LIN {X 0,Y 517.937,Z 91.598,A -85,B 0,C 180,E1 -4909.404,E2 -4909.404} C_VEL
LIN {X 0,Y 516.923,Z 91.726,A -85,B 0,C 180,E1 -4910.052,E2 -4910.052} C_VEL
LIN {X 0,Y 516.851,Z 91.735,A -85,B 0,C 180,E1 -4910.271,E2 -4910.271} C_VEL
LIN {X 0,Y 516.906,Z 91.845,A -85,B 0,C 180,E1 -4911.136,E2 -4911.136} C_VEL
LIN {X 0,Y 518.401,Z 99.769,A -85,B 0,C 180,E1 -4912.604,E2 -4912.604} C_VEL
LIN {X 0,Y 518.069,Z 113.892,A -85,B 0,C 180,E1 -4915.029,E2 -4915.029} C_VEL
LIN {X 0,Y 518.021,Z 116.431,A -85,B 0,C 180,E1 -4915.437,E2 -4915.437} C_VEL
LIN {X 0,Y 520.471,Z 128.644,A -85,B 0,C 180,E1 -4915.705,E2 -4915.705} C_VEL
LIN {X 0,Y 519.69,Z 253.321,A -85,B 0,C 180,E1 -4917.481,E2 -4917.481} C_VEL
LIN {X 0,Y 519.462,Z 267.315,A -85,B 0,C 180,E1 -4917.838,E2 -4917.838} C_VEL
LIN {X 0,Y 519.171,Z 280.563,A -85,B 0,C 180,E1 -4918.326,E2 -4918.326} C_VEL
LIN {X 0,Y 518.764,Z 294.503,A -85,B 0,C 180,E1 -4919.014,E2 -4919.014} C_VEL
LIN {X 0,Y 518.356,Z 306.612,A -85,B 0,C 180,E1 -4919.777,E2 -4919.777} C_VEL
LIN {X 0,Y 517.938,Z 319.149,A -85,B 0,C 180,E1 -4920.758,E2 -4920.758} C_VEL
LIN {X 0,Y 517.552,Z 330.416,A -85,B 0,C 180,E1 -4921.842,E2 -4921.842} C_VEL
LIN {X 0,Y 517.178,Z 339.685,A -85,B 0,C 180,E1 -4922.919,E2 -4922.919} C_VEL
LIN {X 0,Y 516.871,Z 348.845,A -85,B 0,C 180,E1 -4924.207,E2 -4924.207} C_VEL
LIN {X 0,Y 516.661,Z 355.972,A -85,B 0,C 180,E1 -4925.418,E2 -4925.418} C_VEL
LIN {X 0,Y 516.507,Z 362.417,A -85,B 0,C 180,E1 -4926.758,E2 -4926.758} C_VEL
LIN {X 0,Y 516.393,Z 367.484,A -85,B 0,C 180,E1 -4928.075,E2 -4928.075} C_VEL
LIN {X 0,Y 516.349,Z 371.085,A -85,B 0,C 180,E1 -4929.274,E2 -4929.274} C_VEL
LIN {X 0,Y 516.314,Z 373.093,A -85,B 0,C 180,E1 -4930.104,E2 -4930.104} C_VEL
LIN {X 0,Y 516.164,Z 375.912,A -85,B 0,C 180,E1 -4931.749,E2 -4931.749} C_VEL
LIN {X 0,Y 516.203,Z 376.744,A -85,B 0,C 180,E1 -4932.57,E2 -4932.57} C_VEL
LIN {X 0,Y 516.155,Z 377.306,A -85,B 0,C 180,E1 -4934.197,E2 -4934.197} C_VEL
LIN {X 0,Y 516.205,Z 376.454,A -85,B 0,C 180,E1 -4935.813,E2 -4935.813} C_VEL
LIN {X 0,Y 516.269,Z 374.205,A -85,B 0,C 180,E1 -4937.419,E2 -4937.419} C_VEL
LIN {X 0,Y 516.334,Z 370.533,A -85,B 0,C 180,E1 -4939.014,E2 -4939.014} C_VEL
LIN {X 0,Y 516.397,Z 365.356,A -85,B 0,C 180,E1 -4940.6,E2 -4940.6} C_VEL
LIN {X 0,Y 516.526,Z 360.334,A -85,B 0,C 180,E1 -4941.785,E2 -4941.785} C_VEL
LIN {X 0,Y 516.761,Z 353.621,A -85,B 0,C 180,E1 -4943.085,E2 -4943.085} C_VEL
LIN {X 0,Y 516.944,Z 345.726,A -85,B 0,C 180,E1 -4944.342,E2 -4944.342} C_VEL
LIN {X 0,Y 517.288,Z 336.792,A -85,B 0,C 180,E1 -4945.518,E2 -4945.518} C_VEL
LIN {X 0,Y 517.677,Z 326.031,A -85,B 0,C 180,E1 -4946.691,E2 -4946.691} C_VEL
LIN {X 0,Y 518.065,Z 315.147,A -85,B 0,C 180,E1 -4947.666,E2 -4947.666} C_VEL
LIN {X 0,Y 518.475,Z 303.235,A -85,B 0,C 180,E1 -4948.543,E2 -4948.543} C_VEL
LIN {X 0,Y 518.925,Z 289.938,A -85,B 0,C 180,E1 -4949.32,E2 -4949.32} C_VEL
LIN {X 0,Y 519.246,Z 277.171,A -85,B 0,C 180,E1 -4949.902,E2 -4949.902} C_VEL
LIN {X 0,Y 519.516,Z 263.525,A -85,B 0,C 180,E1 -4950.362,E2 -4950.362} C_VEL
LIN {X 0,Y 519.652,Z 249.563,A -85,B 0,C 180,E1 -4950.677,E2 -4950.677} C_VEL
LIN {X 0,Y 520.387,Z 127.623,A -85,B 0,C 180,E1 -4952.399,E2 -4952.399} C_VEL
LIN {X 0,Y 517.972,Z 116.11,A -85,B 0,C 180,E1 -4952.66,E2 -4952.66} C_VEL
LIN {X 0,Y 518.473,Z 99.766,A -85,B 0,C 180,E1 -4955.444,E2 -4955.444} C_VEL
LIN {X 0,Y 516.971,Z 91.715,A -85,B 0,C 180,E1 -4956.925,E2 -4956.925} C_VEL
LIN {X 0,Y 516.932,Z 91.719,A -85,B 0,C 180,E1 -4959.388,E2 -4959.388} C_VEL
LIN {X 0,Y 516.933,Z 91.719,A -85,B 0,C 180,E1 -4962.563,E2 -4962.563} C_VEL
LIN {X 0,Y 516.94,Z 91.715,A -85,B 0,C 180,E1 -4965.161,E2 -4965.161} C_VEL
LIN {X 0,Y 516.893,Z 91.72,A -85,B 0,C 180,E1 -4968.222,E2 -4968.222} C_VEL
LIN {X 0,Y 516.882,Z 91.72,A -85,B 0,C 180,E1 -4970.701,E2 -4970.701} C_VEL
LIN {X 0,Y 516.878,Z 91.726,A -85,B 0,C 180,E1 -4973.222,E2 -4973.222} C_VEL
LIN {X 0,Y 516.917,Z 91.716,A -85,B 0,C 180,E1 -4976.2,E2 -4976.2} C_VEL
LIN {X 0,Y 516.906,Z 91.725,A -85,B 0,C 180,E1 -4979.304,E2 -4979.304} C_VEL
LIN {X 0,Y 516.875,Z 91.722,A -85,B 0,C 180,E1 -4982.548,E2 -4982.548} C_VEL
LIN {X 0,Y 516.884,Z 91.724,A -85,B 0,C 180,E1 -4985.34,E2 -4985.34} C_VEL
LIN {X 0,Y 516.886,Z 91.725,A -85,B 0,C 180,E1 -4988.714,E2 -4988.714} C_VEL
LIN {X 0,Y 516.893,Z 91.719,A -85,B 0,C 180,E1 -4991.775,E2 -4991.775} C_VEL
LIN {X 0,Y 516.889,Z 91.724,A -85,B 0,C 180,E1 -4995.012,E2 -4995.012} C_VEL
LIN {X 0,Y 516.886,Z 91.721,A -85,B 0,C 180,E1 -4997.24,E2 -4997.24} C_VEL
LIN {X 0,Y 516.905,Z 91.722,A -85,B 0,C 180,E1 -5000.286,E2 -5000.286} C_VEL
LIN {X 0,Y 516.862,Z 91.723,A -85,B 0,C 180,E1 -5003.343,E2 -5003.343} C_VEL
LIN {X 0,Y 516.888,Z 91.724,A -85,B 0,C 180,E1 -5006.124,E2 -5006.124} C_VEL
LIN {X 0,Y 516.871,Z 91.723,A -85,B 0,C 180,E1 -5008.937,E2 -5008.937} C_VEL
LIN {X 0,Y 516.901,Z 91.719,A -85,B 0,C 180,E1 -5011.588,E2 -5011.588} C_VEL
LIN {X 0,Y 516.915,Z 91.724,A -85,B 0,C 180,E1 -5014.214,E2 -5014.214} C_VEL
LIN {X 0,Y 516.888,Z 91.72,A -85,B 0,C 180,E1 -5016.781,E2 -5016.781} C_VEL
LIN {X 0,Y 516.919,Z 91.721,A -85,B 0,C 180,E1 -5019.734,E2 -5019.734} C_VEL
LIN {X 0,Y 516.913,Z 91.717,A -85,B 0,C 180,E1 -5022.599,E2 -5022.599} C_VEL
LIN {X 0,Y 516.924,Z 91.715,A -85,B 0,C 180,E1 -5025.033,E2 -5025.033} C_VEL
LIN {X 0,Y 516.988,Z 91.709,A -85,B 0,C 180,E1 -5028.237,E2 -5028.237} C_VEL
LIN {X 0,Y 516.96,Z 91.716,A -85,B 0,C 180,E1 -5031.402,E2 -5031.402} C_VEL
LIN {X 0,Y 517.034,Z 91.701,A -85,B 0,C 180,E1 -5034.543,E2 -5034.543} C_VEL
LIN {X 0,Y 517.074,Z 91.701,A -85,B 0,C 180,E1 -5037.666,E2 -5037.666} C_VEL
LIN {X 0,Y 517.087,Z 91.696,A -85,B 0,C 180,E1 -5040.781,E2 -5040.781} C_VEL
LIN {X 0,Y 517.008,Z 91.711,A -85,B 0,C 180,E1 -5043.119,E2 -5043.119} C_VEL
LIN {X 0,Y 517.002,Z 91.705,A -85,B 0,C 180,E1 -5046.246,E2 -5046.246} C_VEL
LIN {X 0,Y 516.947,Z 91.716,A -85,B 0,C 180,E1 -5049.392,E2 -5049.392} C_VEL
LIN {X 0,Y 516.945,Z 91.712,A -85,B 0,C 180,E1 -5051.81,E2 -5051.81} C_VEL
LIN {X 0,Y 516.938,Z 91.718,A -85,B 0,C 180,E1 -5055.149,E2 -5055.149} C_VEL
LIN {X 0,Y 516.92,Z 91.717,A -85,B 0,C 180,E1 -5058.224,E2 -5058.224} C_VEL
LIN {X 0,Y 516.907,Z 91.726,A -85,B 0,C 180,E1 -5060.704,E2 -5060.704} C_VEL
LIN {X 0,Y 516.907,Z 91.719,A -85,B 0,C 180,E1 -5064.074,E2 -5064.074} C_VEL
LIN {X 0,Y 516.926,Z 91.721,A -85,B 0,C 180,E1 -5066.66,E2 -5066.66} C_VEL
LIN {X 0,Y 516.908,Z 91.717,A -85,B 0,C 180,E1 -5069.526,E2 -5069.526} C_VEL
LIN {X 0,Y 516.895,Z 91.724,A -85,B 0,C 180,E1 -5072.546,E2 -5072.546} C_VEL
LIN {X 0,Y 516.876,Z 91.721,A -85,B 0,C 180,E1 -5075.334,E2 -5075.334} C_VEL
LIN {X 0,Y 516.878,Z 91.726,A -85,B 0,C 180,E1 -5077.945,E2 -5077.945} C_VEL
LIN {X 0,Y 516.882,Z 91.721,A -85,B 0,C 180,E1 -5080.743,E2 -5080.743} C_VEL
LIN {X 0,Y 516.883,Z 91.72,A -85,B 0,C 180,E1 -5082.833,E2 -5082.833} C_VEL
LIN {X 0,Y 516.922,Z 91.715,A -85,B 0,C 180,E1 -5085.012,E2 -5085.012} C_VEL
LIN {X 0,Y 516.914,Z 91.718,A -85,B 0,C 180,E1 -5088.4,E2 -5088.4} C_VEL
LIN {X 0,Y 516.88,Z 91.723,A -85,B 0,C 180,E1 -5091.286,E2 -5091.286} C_VEL
LIN {X 0,Y 516.871,Z 91.723,A -85,B 0,C 180,E1 -5094.221,E2 -5094.221} C_VEL
LIN {X 0,Y 516.895,Z 91.721,A -85,B 0,C 180,E1 -5097.055,E2 -5097.055} C_VEL
LIN {X 0,Y 516.887,Z 91.726,A -85,B 0,C 180,E1 -5099.797,E2 -5099.797} C_VEL
LIN {X 0,Y 516.926,Z 91.719,A -85,B 0,C 180,E1 -5102.469,E2 -5102.469} C_VEL
LIN {X 0,Y 516.957,Z 91.852,A -85,B 0,C 180,E1 -5103.888,E2 -5103.888} C_VEL
LIN {X 0,Y 519.076,Z 102.657,A -85,B 0,C 180,E1 -5105.611,E2 -5105.611} C_VEL
LIN {X 0,Y 518.535,Z 121.144,A -85,B 0,C 180,E1 -5108.327,E2 -5108.327} C_VEL
LIN {X 0,Y 517.999,Z 142.503,A -85,B 0,C 180,E1 -5111.381,E2 -5111.381} C_VEL
LIN {X 0,Y 520.393,Z 156.779,A -85,B 0,C 180,E1 -5111.672,E2 -5111.672} C_VEL
LIN {X 0,Y 519.58,Z 280.355,A -85,B 0,C 180,E1 -5113.423,E2 -5113.423} C_VEL
LIN {X 0,Y 519.338,Z 294.907,A -85,B 0,C 180,E1 -5113.792,E2 -5113.792} C_VEL
LIN {X 0,Y 519.05,Z 308.369,A -85,B 0,C 180,E1 -5114.289,E2 -5114.289} C_VEL
LIN {X 0,Y 518.646,Z 320.6,A -85,B 0,C 180,E1 -5114.881,E2 -5114.881} C_VEL
LIN {X 0,Y 518.226,Z 333.464,A -85,B 0,C 180,E1 -5115.672,E2 -5115.672} C_VEL
LIN {X 0,Y 517.779,Z 345.158,A -85,B 0,C 180,E1 -5116.56,E2 -5116.56} C_VEL
LIN {X 0,Y 517.474,Z 354.895,A -85,B 0,C 180,E1 -5117.451,E2 -5117.451} C_VEL
LIN {X 0,Y 517.116,Z 365.679,A -85,B 0,C 180,E1 -5118.636,E2 -5118.636} C_VEL
LIN {X 0,Y 516.817,Z 374.585,A -85,B 0,C 180,E1 -5119.819,E2 -5119.819} C_VEL
LIN {X 0,Y 516.607,Z 383.12,A -85,B 0,C 180,E1 -5121.198,E2 -5121.198} C_VEL
LIN {X 0,Y 516.443,Z 389.998,A -85,B 0,C 180,E1 -5122.573,E2 -5122.573} C_VEL
LIN {X 0,Y 516.352,Z 396.142,A -85,B 0,C 180,E1 -5124.142,E2 -5124.142} C_VEL
LIN {X 0,Y 516.262,Z 399.65,A -85,B 0,C 180,E1 -5125.316,E2 -5125.316} C_VEL
LIN {X 0,Y 516.325,Z 401.539,A -85,B 0,C 180,E1 -5126.099,E2 -5126.099} C_VEL
LIN {X 0,Y 516.26,Z 404.245,A -85,B 0,C 180,E1 -5127.661,E2 -5127.661} C_VEL
LIN {X 0,Y 516.158,Z 405.582,A -85,B 0,C 180,E1 -5129.221,E2 -5129.221} C_VEL
LIN {X 0,Y 516.158,Z 405.579,A -85,B 0,C 180,E1 -5130.781,E2 -5130.781} C_VEL
LIN {X 0,Y 516.261,Z 404.237,A -85,B 0,C 180,E1 -5132.342,E2 -5132.342} C_VEL
LIN {X 0,Y 516.325,Z 401.526,A -85,B 0,C 180,E1 -5133.904,E2 -5133.904} C_VEL
LIN {X 0,Y 516.354,Z 397.368,A -85,B 0,C 180,E1 -5135.468,E2 -5135.468} C_VEL
LIN {X 0,Y 516.405,Z 391.641,A -85,B 0,C 180,E1 -5137.037,E2 -5137.037} C_VEL
LIN {X 0,Y 516.562,Z 385.188,A -85,B 0,C 180,E1 -5138.411,E2 -5138.411} C_VEL
LIN {X 0,Y 516.752,Z 377.171,A -85,B 0,C 180,E1 -5139.789,E2 -5139.789} C_VEL
LIN {X 0,Y 517.05,Z 368.787,A -85,B 0,C 180,E1 -5140.971,E2 -5140.971} C_VEL
LIN {X 0,Y 517.371,Z 358.473,A -85,B 0,C 180,E1 -5142.18,E2 -5142.18} C_VEL
LIN {X 0,Y 517.722,Z 347.43,A -85,B 0,C 180,E1 -5143.244,E2 -5143.244} C_VEL
LIN {X 0,Y 518.078,Z 336.228,A -85,B 0,C 180,E1 -5144.134,E2 -5144.134} C_VEL
LIN {X 0,Y 518.512,Z 324.028,A -85,B 0,C 180,E1 -5144.925,E2 -5144.925} C_VEL
LIN {X 0,Y 518.956,Z 310.488,A -85,B 0,C 180,E1 -5145.615,E2 -5145.615} C_VEL
LIN {X 0,Y 519.26,Z 296.705,A -85,B 0,C 180,E1 -5146.147,E2 -5146.147} C_VEL
LIN {X 0,Y 519.549,Z 282.425,A -85,B 0,C 180,E1 -5146.53,E2 -5146.53} C_VEL
LIN {X 0,Y 519.768,Z 258.348,A -85,B 0,C 180,E1 -5146.902,E2 -5146.902} C_VEL
LIN {X 0,Y 520.277,Z 155.65,A -85,B 0,C 180,E1 -5148.347,E2 -5148.347} C_VEL
LIN {X 0,Y 517.932,Z 142.086,A -85,B 0,C 180,E1 -5148.637,E2 -5148.637} C_VEL
LIN {X 0,Y 518.551,Z 121.098,A -85,B 0,C 180,E1 -5151.675,E2 -5151.675} C_VEL
LIN {X 0,Y 519.092,Z 102.719,A -85,B 0,C 180,E1 -5154.391,E2 -5154.391} C_VEL
LIN {X 0,Y 517.157,Z 92.942,A -85,B 0,C 180,E1 -5155.975,E2 -5155.975} C_VEL
LIN {X 0,Y 516.91,Z 91.724,A -85,B 0,C 180,E1 -5156.187,E2 -5156.187} C_VEL
LIN {X 0,Y 516.925,Z 91.723,A -85,B 0,C 180,E1 -5158.416,E2 -5158.416} C_VEL
LIN {X 0,Y 516.898,Z 91.724,A -85,B 0,C 180,E1 -5161.11,E2 -5161.11} C_VEL
LIN {X 0,Y 516.897,Z 91.727,A -85,B 0,C 180,E1 -5163.963,E2 -5163.963} C_VEL
LIN {X 0,Y 516.864,Z 91.724,A -85,B 0,C 180,E1 -5166.748,E2 -5166.748} C_VEL
LIN {X 0,Y 516.883,Z 91.726,A -85,B 0,C 180,E1 -5169.722,E2 -5169.722} C_VEL
LIN {X 0,Y 516.918,Z 91.72,A -85,B 0,C 180,E1 -5171.776,E2 -5171.776} C_VEL
LIN {X 0,Y 516.908,Z 91.718,A -85,B 0,C 180,E1 -5175.007,E2 -5175.007} C_VEL
LIN {X 0,Y 516.926,Z 91.71,A -85,B 0,C 180,E1 -5178.399,E2 -5178.399} C_VEL
LIN {X 0,Y 516.889,Z 91.724,A -85,B 0,C 180,E1 -5181.283,E2 -5181.283} C_VEL
LIN {X 0,Y 516.88,Z 91.722,A -85,B 0,C 180,E1 -5184.219,E2 -5184.219} C_VEL
LIN {X 0,Y 516.894,Z 91.722,A -85,B 0,C 180,E1 -5187.051,E2 -5187.051} C_VEL
LIN {X 0,Y 516.896,Z 91.722,A -85,B 0,C 180,E1 -5189.795,E2 -5189.795} C_VEL
LIN {X 0,Y 516.906,Z 91.716,A -85,B 0,C 180,E1 -5192.464,E2 -5192.464} C_VEL
LIN {X 0,Y 516.878,Z 91.728,A -85,B 0,C 180,E1 -5195.068,E2 -5195.068} C_VEL
LIN {X 0,Y 516.882,Z 91.722,A -85,B 0,C 180,E1 -5197.62,E2 -5197.62} C_VEL
LIN {X 0,Y 516.942,Z 91.71,A -85,B 0,C 180,E1 -5200.128,E2 -5200.128} C_VEL
LIN {X 0,Y 516.907,Z 91.723,A -85,B 0,C 180,E1 -5202.593,E2 -5202.593} C_VEL
LIN {X 0,Y 516.947,Z 91.717,A -85,B 0,C 180,E1 -5205.028,E2 -5205.028} C_VEL
LIN {X 0,Y 516.978,Z 91.711,A -85,B 0,C 180,E1 -5208.232,E2 -5208.232} C_VEL
LIN {X 0,Y 516.963,Z 91.71,A -85,B 0,C 180,E1 -5211.397,E2 -5211.397} C_VEL
LIN {X 0,Y 517.021,Z 91.709,A -85,B 0,C 180,E1 -5214.538,E2 -5214.538} C_VEL
LIN {X 0,Y 517.088,Z 91.694,A -85,B 0,C 180,E1 -5217.661,E2 -5217.661} C_VEL
LIN {X 0,Y 517.096,Z 91.692,A -85,B 0,C 180,E1 -5220.776,E2 -5220.776} C_VEL
LIN {X 0,Y 516.988,Z 91.708,A -85,B 0,C 180,E1 -5223.114,E2 -5223.114} C_VEL
LIN {X 0,Y 516.993,Z 91.711,A -85,B 0,C 180,E1 -5226.241,E2 -5226.241} C_VEL
LIN {X 0,Y 516.944,Z 91.715,A -85,B 0,C 180,E1 -5229.386,E2 -5229.386} C_VEL
LIN {X 0,Y 516.954,Z 91.718,A -85,B 0,C 180,E1 -5231.804,E2 -5231.804} C_VEL
LIN {X 0,Y 516.943,Z 91.716,A -85,B 0,C 180,E1 -5235.142,E2 -5235.142} C_VEL
LIN {X 0,Y 516.91,Z 91.718,A -85,B 0,C 180,E1 -5238.219,E2 -5238.219} C_VEL
LIN {X 0,Y 516.901,Z 91.718,A -85,B 0,C 180,E1 -5240.698,E2 -5240.698} C_VEL
LIN {X 0,Y 516.88,Z 91.721,A -85,B 0,C 180,E1 -5244.07,E2 -5244.07} C_VEL
LIN {X 0,Y 516.9,Z 91.72,A -85,B 0,C 180,E1 -5246.655,E2 -5246.655} C_VEL
LIN {X 0,Y 516.899,Z 91.715,A -85,B 0,C 180,E1 -5249.52,E2 -5249.52} C_VEL
LIN {X 0,Y 516.882,Z 91.725,A -85,B 0,C 180,E1 -5252.539,E2 -5252.539} C_VEL
LIN {X 0,Y 516.852,Z 91.728,A -85,B 0,C 180,E1 -5255.326,E2 -5255.326} C_VEL
LIN {X 0,Y 516.863,Z 91.721,A -85,B 0,C 180,E1 -5257.939,E2 -5257.939} C_VEL
LIN {X 0,Y 516.867,Z 91.727,A -85,B 0,C 180,E1 -5260.738,E2 -5260.738} C_VEL
LIN {X 0,Y 516.864,Z 91.729,A -85,B 0,C 180,E1 -5262.828,E2 -5262.828} C_VEL
LIN {X 0,Y 516.875,Z 91.724,A -85,B 0,C 180,E1 -5265.004,E2 -5265.004} C_VEL
LIN {X 0,Y 516.88,Z 91.731,A -85,B 0,C 180,E1 -5268.397,E2 -5268.397} C_VEL
LIN {X 0,Y 516.851,Z 91.735,A -85,B 0,C 180,E1 -5270.271,E2 -5270.271} C_VEL
LIN {X 0,Y 516.63,Z 92.161,A -85,B 0,C 180,E1 -5270.7,E2 -5270.7} C_VEL
LIN {X 0,Y 516.043,Z 93.272,A -85,B 0,C 180,E1 -5271.112,E2 -5271.112} C_VEL
LIN {X 0,Y 514.758,Z 95.823,A -85,B 0,C 180,E1 -5271.695,E2 -5271.695} C_VEL
LIN {X 0,Y 511.765,Z 103.822,A -85,B 0,C 180,E1 -5272.982,E2 -5272.982} C_VEL
LIN {X 0,Y 511.44,Z 106.048,A -85,B 0,C 180,E1 -5273.361,E2 -5273.361} C_VEL
LIN {X 0,Y 511.096,Z 116.359,A -85,B 0,C 180,E1 -5275.149,E2 -5275.149} C_VEL
LIN {X 0,Y 513.748,Z 129.088,A -85,B 0,C 180,E1 -5275.457,E2 -5275.457} C_VEL
LIN {X 0,Y 512.927,Z 252.499,A -85,B 0,C 180,E1 -5277.232,E2 -5277.232} C_VEL
LIN {X 0,Y 512.654,Z 267.254,A -85,B 0,C 180,E1 -5277.606,E2 -5277.606} C_VEL
LIN {X 0,Y 512.346,Z 280.832,A -85,B 0,C 180,E1 -5278.113,E2 -5278.113} C_VEL
LIN {X 0,Y 511.918,Z 294.283,A -85,B 0,C 180,E1 -5278.783,E2 -5278.783} C_VEL
LIN {X 0,Y 511.462,Z 307.149,A -85,B 0,C 180,E1 -5279.605,E2 -5279.605} C_VEL
LIN {X 0,Y 511.042,Z 319.053,A -85,B 0,C 180,E1 -5280.55,E2 -5280.55} C_VEL
LIN {X 0,Y 510.64,Z 329.18,A -85,B 0,C 180,E1 -5281.525,E2 -5281.525} C_VEL
LIN {X 0,Y 510.19,Z 339.675,A -85,B 0,C 180,E1 -5282.739,E2 -5282.739} C_VEL
LIN {X 0,Y 509.867,Z 348.887,A -85,B 0,C 180,E1 -5284.045,E2 -5284.045} C_VEL
LIN {X 0,Y 509.615,Z 356.504,A -85,B 0,C 180,E1 -5285.365,E2 -5285.365} C_VEL
LIN {X 0,Y 509.432,Z 363.378,A -85,B 0,C 180,E1 -5286.846,E2 -5286.846} C_VEL
LIN {X 0,Y 509.319,Z 368.114,A -85,B 0,C 180,E1 -5288.125,E2 -5288.125} C_VEL
LIN {X 0,Y 509.233,Z 372.697,A -85,B 0,C 180,E1 -5289.785,E2 -5289.785} C_VEL
LIN {X 0,Y 509.087,Z 375.784,A -85,B 0,C 180,E1 -5291.486,E2 -5291.486} C_VEL
LIN {X 0,Y 509.08,Z 377.3,A -85,B 0,C 180,E1 -5293.146,E2 -5293.146} C_VEL
LIN {X 0,Y 509.091,Z 377.376,A -85,B 0,C 180,E1 -5294.793,E2 -5294.793} C_VEL
LIN {X 0,Y 509.108,Z 376.02,A -85,B 0,C 180,E1 -5296.426,E2 -5296.426} C_VEL
LIN {X 0,Y 509.205,Z 373.247,A -85,B 0,C 180,E1 -5298.051,E2 -5298.051} C_VEL
LIN {X 0,Y 509.291,Z 369.024,A -85,B 0,C 180,E1 -5299.664,E2 -5299.664} C_VEL
LIN {X 0,Y 509.418,Z 363.242,A -85,B 0,C 180,E1 -5301.27,E2 -5301.27} C_VEL
LIN {X 0,Y 509.621,Z 356.741,A -85,B 0,C 180,E1 -5302.67,E2 -5302.67} C_VEL
LIN {X 0,Y 509.885,Z 348.713,A -85,B 0,C 180,E1 -5304.065,E2 -5304.065} C_VEL
LIN {X 0,Y 510.187,Z 340.337,A -85,B 0,C 180,E1 -5305.258,E2 -5305.258} C_VEL
LIN {X 0,Y 510.597,Z 330.264,A -85,B 0,C 180,E1 -5306.448,E2 -5306.448} C_VEL
LIN {X 0,Y 510.983,Z 319.057,A -85,B 0,C 180,E1 -5307.536,E2 -5307.536} C_VEL
LIN {X 0,Y 511.402,Z 307.943,A -85,B 0,C 180,E1 -5308.424,E2 -5308.424} C_VEL
LIN {X 0,Y 511.893,Z 295.811,A -85,B 0,C 180,E1 -5309.212,E2 -5309.212} C_VEL
LIN {X 0,Y 512.29,Z 282.406,A -85,B 0,C 180,E1 -5309.901,E2 -5309.901} C_VEL
LIN {X 0,Y 512.615,Z 268.364,A -85,B 0,C 180,E1 -5310.441,E2 -5310.441} C_VEL
LIN {X 0,Y 512.823,Z 254.558,A -85,B 0,C 180,E1 -5310.809,E2 -5310.809} C_VEL
LIN {X 0,Y 513.055,Z 227.07,A -85,B 0,C 180,E1 -5311.231,E2 -5311.231} C_VEL
LIN {X 0,Y 513.653,Z 128.738,A -85,B 0,C 180,E1 -5312.633,E2 -5312.633} C_VEL
LIN {X 0,Y 511.048,Z 116.22,A -85,B 0,C 180,E1 -5312.931,E2 -5312.931} C_VEL
LIN {X 0,Y 511.553,Z 101.194,A -85,B 0,C 180,E1 -5315.517,E2 -5315.517} C_VEL
LIN {X 0,Y 509.951,Z 92.59,A -85,B 0,C 180,E1 -5317.124,E2 -5317.124} C_VEL
LIN {X 0,Y 509.874,Z 92.6,A -85,B 0,C 180,E1 -5319.52,E2 -5319.52} C_VEL
LIN {X 0,Y 509.912,Z 92.598,A -85,B 0,C 180,E1 -5321.93,E2 -5321.93} C_VEL
LIN {X 0,Y 509.905,Z 92.592,A -85,B 0,C 180,E1 -5325.263,E2 -5325.263} C_VEL
LIN {X 0,Y 509.873,Z 92.596,A -85,B 0,C 180,E1 -5328.01,E2 -5328.01} C_VEL
LIN {X 0,Y 509.827,Z 92.601,A -85,B 0,C 180,E1 -5331.001,E2 -5331.001} C_VEL
LIN {X 0,Y 509.834,Z 92.605,A -85,B 0,C 180,E1 -5333.562,E2 -5333.562} C_VEL
LIN {X 0,Y 509.885,Z 92.592,A -85,B 0,C 180,E1 -5336.382,E2 -5336.382} C_VEL
LIN {X 0,Y 509.854,Z 92.599,A -85,B 0,C 180,E1 -5338.844,E2 -5338.844} C_VEL
LIN {X 0,Y 509.804,Z 92.605,A -85,B 0,C 180,E1 -5341.59,E2 -5341.59} C_VEL
LIN {X 0,Y 509.833,Z 92.599,A -85,B 0,C 180,E1 -5344.413,E2 -5344.413} C_VEL
LIN {X 0,Y 509.799,Z 92.606,A -85,B 0,C 180,E1 -5347.341,E2 -5347.341} C_VEL
LIN {X 0,Y 509.856,Z 92.597,A -85,B 0,C 180,E1 -5350.379,E2 -5350.379} C_VEL
LIN {X 0,Y 509.824,Z 92.604,A -85,B 0,C 180,E1 -5353.068,E2 -5353.068} C_VEL
LIN {X 0,Y 509.849,Z 92.596,A -85,B 0,C 180,E1 -5355.788,E2 -5355.788} C_VEL
LIN {X 0,Y 509.842,Z 92.605,A -85,B 0,C 180,E1 -5358.578,E2 -5358.578} C_VEL
LIN {X 0,Y 509.833,Z 92.598,A -85,B 0,C 180,E1 -5361.665,E2 -5361.665} C_VEL
LIN {X 0,Y 509.823,Z 92.606,A -85,B 0,C 180,E1 -5364.626,E2 -5364.626} C_VEL
LIN {X 0,Y 509.843,Z 92.597,A -85,B 0,C 180,E1 -5367.484,E2 -5367.484} C_VEL
LIN {X 0,Y 509.856,Z 92.604,A -85,B 0,C 180,E1 -5370.271,E2 -5370.271} C_VEL
LIN {X 0,Y 509.866,Z 92.595,A -85,B 0,C 180,E1 -5372.947,E2 -5372.947} C_VEL
LIN {X 0,Y 509.875,Z 92.595,A -85,B 0,C 180,E1 -5375.578,E2 -5375.578} C_VEL
LIN {X 0,Y 509.835,Z 92.605,A -85,B 0,C 180,E1 -5378.153,E2 -5378.153} C_VEL
LIN {X 0,Y 509.846,Z 92.597,A -85,B 0,C 180,E1 -5380.684,E2 -5380.684} C_VEL
LIN {X 0,Y 509.87,Z 92.594,A -85,B 0,C 180,E1 -5383.178,E2 -5383.178} C_VEL
LIN {X 0,Y 509.849,Z 92.603,A -85,B 0,C 180,E1 -5385.637,E2 -5385.637} C_VEL
LIN {X 0,Y 509.911,Z 92.589,A -85,B 0,C 180,E1 -5388.878,E2 -5388.878} C_VEL
LIN {X 0,Y 509.939,Z 92.587,A -85,B 0,C 180,E1 -5392.081,E2 -5392.081} C_VEL
LIN {X 0,Y 509.983,Z 92.579,A -85,B 0,C 180,E1 -5394.467,E2 -5394.467} C_VEL
LIN {X 0,Y 510.045,Z 92.577,A -85,B 0,C 180,E1 -5397.634,E2 -5397.634} C_VEL
LIN {X 0,Y 510.057,Z 92.572,A -85,B 0,C 180,E1 -5400.792,E2 -5400.792} C_VEL
LIN {X 0,Y 509.95,Z 92.591,A -85,B 0,C 180,E1 -5403.163,E2 -5403.163} C_VEL
LIN {X 0,Y 509.97,Z 92.581,A -85,B 0,C 180,E1 -5406.332,E2 -5406.332} C_VEL
LIN {X 0,Y 509.909,Z 92.592,A -85,B 0,C 180,E1 -5408.723,E2 -5408.723} C_VEL
LIN {X 0,Y 509.897,Z 92.59,A -85,B 0,C 180,E1 -5411.934,E2 -5411.934} C_VEL
LIN {X 0,Y 509.887,Z 92.595,A -85,B 0,C 180,E1 -5415.244,E2 -5415.244} C_VEL
LIN {X 0,Y 509.883,Z 92.592,A -85,B 0,C 180,E1 -5418.003,E2 -5418.003} C_VEL
LIN {X 0,Y 509.845,Z 92.601,A -85,B 0,C 180,E1 -5421.004,E2 -5421.004} C_VEL
LIN {X 0,Y 509.833,Z 92.598,A -85,B 0,C 180,E1 -5423.565,E2 -5423.565} C_VEL
LIN {X 0,Y 509.91,Z 92.595,A -85,B 0,C 180,E1 -5426.381,E2 -5426.381} C_VEL
LIN {X 0,Y 509.874,Z 92.596,A -85,B 0,C 180,E1 -5428.846,E2 -5428.846} C_VEL
LIN {X 0,Y 509.818,Z 92.6,A -85,B 0,C 180,E1 -5431.592,E2 -5431.592} C_VEL
LIN {X 0,Y 509.849,Z 92.603,A -85,B 0,C 180,E1 -5434.415,E2 -5434.415} C_VEL
LIN {X 0,Y 509.816,Z 92.6,A -85,B 0,C 180,E1 -5437.343,E2 -5437.343} C_VEL
LIN {X 0,Y 509.836,Z 92.602,A -85,B 0,C 180,E1 -5440.384,E2 -5440.384} C_VEL
LIN {X 0,Y 509.823,Z 92.599,A -85,B 0,C 180,E1 -5443.064,E2 -5443.064} C_VEL
LIN {X 0,Y 509.83,Z 92.605,A -85,B 0,C 180,E1 -5445.794,E2 -5445.794} C_VEL
LIN {X 0,Y 509.856,Z 92.596,A -85,B 0,C 180,E1 -5448.576,E2 -5448.576} C_VEL
LIN {X 0,Y 509.85,Z 92.604,A -85,B 0,C 180,E1 -5451.788,E2 -5451.788} C_VEL
LIN {X 0,Y 509.829,Z 92.599,A -85,B 0,C 180,E1 -5454.624,E2 -5454.624} C_VEL
LIN {X 0,Y 509.861,Z 92.602,A -85,B 0,C 180,E1 -5457.482,E2 -5457.482} C_VEL
LIN {X 0,Y 509.859,Z 92.599,A -85,B 0,C 180,E1 -5460.275,E2 -5460.275} C_VEL
LIN {X 0,Y 509.884,Z 92.599,A -85,B 0,C 180,E1 -5462.946,E2 -5462.946} C_VEL
LIN {X 0,Y 509.917,Z 92.679,A -85,B 0,C 180,E1 -5463.666,E2 -5463.666} C_VEL
LIN {X 0,Y 512.18,Z 104.13,A -85,B 0,C 180,E1 -5465.522,E2 -5465.522} C_VEL
LIN {X 0,Y 511.591,Z 122.365,A -85,B 0,C 180,E1 -5468.229,E2 -5468.229} C_VEL
LIN {X 0,Y 511.024,Z 142.06,A -85,B 0,C 180,E1 -5471.115,E2 -5471.115} C_VEL
LIN {X 0,Y 513.642,Z 158.145,A -85,B 0,C 180,E1 -5471.447,E2 -5471.447} C_VEL
LIN {X 0,Y 512.784,Z 280.074,A -85,B 0,C 180,E1 -5473.197,E2 -5473.197} C_VEL
LIN {X 0,Y 512.527,Z 294.484,A -85,B 0,C 180,E1 -5473.565,E2 -5473.565} C_VEL
LIN {X 0,Y 512.188,Z 308.147,A -85,B 0,C 180,E1 -5474.073,E2 -5474.073} C_VEL
LIN {X 0,Y 511.71,Z 322.154,A -85,B 0,C 180,E1 -5474.773,E2 -5474.773} C_VEL
LIN {X 0,Y 511.26,Z 334.683,A -85,B 0,C 180,E1 -5475.574,E2 -5475.574} C_VEL
LIN {X 0,Y 510.774,Z 346.128,A -85,B 0,C 180,E1 -5476.474,E2 -5476.474} C_VEL
LIN {X 0,Y 510.43,Z 356.845,A -85,B 0,C 180,E1 -5477.497,E2 -5477.497} C_VEL
LIN {X 0,Y 510.08,Z 367.112,A -85,B 0,C 180,E1 -5478.678,E2 -5478.678} C_VEL
LIN {X 0,Y 509.726,Z 375.745,A -85,B 0,C 180,E1 -5479.876,E2 -5479.876} C_VEL
LIN {X 0,Y 509.518,Z 384.016,A -85,B 0,C 180,E1 -5481.274,E2 -5481.274} C_VEL
LIN {X 0,Y 509.367,Z 389.8,A -85,B 0,C 180,E1 -5482.469,E2 -5482.469} C_VEL
LIN {X 0,Y 509.262,Z 394.543,A -85,B 0,C 180,E1 -5483.663,E2 -5483.663} C_VEL
LIN {X 0,Y 509.233,Z 398.385,A -85,B 0,C 180,E1 -5484.854,E2 -5484.854} C_VEL
LIN {X 0,Y 509.217,Z 401.343,A -85,B 0,C 180,E1 -5486.044,E2 -5486.044} C_VEL
LIN {X 0,Y 509.189,Z 404.05,A -85,B 0,C 180,E1 -5487.628,E2 -5487.628} C_VEL
LIN {X 0,Y 509.071,Z 405.388,A -85,B 0,C 180,E1 -5489.21,E2 -5489.21} C_VEL
LIN {X 0,Y 509.071,Z 405.384,A -85,B 0,C 180,E1 -5490.792,E2 -5490.792} C_VEL
LIN {X 0,Y 509.189,Z 404.041,A -85,B 0,C 180,E1 -5492.374,E2 -5492.374} C_VEL
LIN {X 0,Y 509.218,Z 401.327,A -85,B 0,C 180,E1 -5493.958,E2 -5493.958} C_VEL
LIN {X 0,Y 509.265,Z 397.167,A -85,B 0,C 180,E1 -5495.545,E2 -5495.545} C_VEL
LIN {X 0,Y 509.33,Z 391.439,A -85,B 0,C 180,E1 -5497.135,E2 -5497.135} C_VEL
LIN {X 0,Y 509.487,Z 384.983,A -85,B 0,C 180,E1 -5498.529,E2 -5498.529} C_VEL
LIN {X 0,Y 509.708,Z 376.963,A -85,B 0,C 180,E1 -5499.926,E2 -5499.926} C_VEL
LIN {X 0,Y 510.017,Z 368.576,A -85,B 0,C 180,E1 -5501.124,E2 -5501.124} C_VEL
LIN {X 0,Y 510.378,Z 357.836,A -85,B 0,C 180,E1 -5502.396,E2 -5502.396} C_VEL
LIN {X 0,Y 510.745,Z 347.21,A -85,B 0,C 180,E1 -5503.428,E2 -5503.428} C_VEL
LIN {X 0,Y 511.208,Z 334.574,A -85,B 0,C 180,E1 -5504.43,E2 -5504.43} C_VEL
LIN {X 0,Y 511.71,Z 322.04,A -85,B 0,C 180,E1 -5505.23,E2 -5505.23} C_VEL
LIN {X 0,Y 512.172,Z 308.022,A -85,B 0,C 180,E1 -5505.93,E2 -5505.93} C_VEL
LIN {X 0,Y 512.48,Z 294.588,A -85,B 0,C 180,E1 -5506.432,E2 -5506.432} C_VEL
LIN {X 0,Y 512.794,Z 279.998,A -85,B 0,C 180,E1 -5506.805,E2 -5506.805} C_VEL
LIN {X 0,Y 513.613,Z 157.4,A -85,B 0,C 180,E1 -5508.569,E2 -5508.569} C_VEL
LIN {X 0,Y 511.028,Z 141.837,A -85,B 0,C 180,E1 -5508.909,E2 -5508.909} C_VEL
LIN {X 0,Y 511.649,Z 120.973,A -85,B 0,C 180,E1 -5511.982,E2 -5511.982} C_VEL
LIN {X 0,Y 512.242,Z 104.333,A -85,B 0,C 180,E1 -5514.477,E2 -5514.477} C_VEL
LIN {X 0,Y 509.871,Z 92.6,A -85,B 0,C 180,E1 -5516.43,E2 -5516.43} C_VEL
LIN {X 0,Y 509.884,Z 92.598,A -85,B 0,C 180,E1 -5518.845,E2 -5518.845} C_VEL
LIN {X 0,Y 509.829,Z 92.604,A -85,B 0,C 180,E1 -5521.591,E2 -5521.591} C_VEL
LIN {X 0,Y 509.849,Z 92.603,A -85,B 0,C 180,E1 -5524.415,E2 -5524.415} C_VEL
LIN {X 0,Y 509.819,Z 92.6,A -85,B 0,C 180,E1 -5527.342,E2 -5527.342} C_VEL
LIN {X 0,Y 509.849,Z 92.599,A -85,B 0,C 180,E1 -5530.382,E2 -5530.382} C_VEL
LIN {X 0,Y 509.813,Z 92.602,A -85,B 0,C 180,E1 -5533.059,E2 -5533.059} C_VEL
LIN {X 0,Y 509.835,Z 92.605,A -85,B 0,C 180,E1 -5535.793,E2 -5535.793} C_VEL
LIN {X 0,Y 509.868,Z 92.587,A -85,B 0,C 180,E1 -5538.574,E2 -5538.574} C_VEL
LIN {X 0,Y 509.862,Z 92.6,A -85,B 0,C 180,E1 -5541.786,E2 -5541.786} C_VEL
LIN {X 0,Y 509.839,Z 92.598,A -85,B 0,C 180,E1 -5544.621,E2 -5544.621} C_VEL
LIN {X 0,Y 509.873,Z 92.601,A -85,B 0,C 180,E1 -5547.48,E2 -5547.48} C_VEL
LIN {X 0,Y 509.871,Z 92.594,A -85,B 0,C 180,E1 -5550.273,E2 -5550.273} C_VEL
LIN {X 0,Y 509.888,Z 92.595,A -85,B 0,C 180,E1 -5553.629,E2 -5553.629} C_VEL
LIN {X 0,Y 509.834,Z 92.597,A -85,B 0,C 180,E1 -5556.435,E2 -5556.435} C_VEL
LIN {X 0,Y 509.927,Z 92.584,A -85,B 0,C 180,E1 -5559.843,E2 -5559.843} C_VEL
LIN {X 0,Y 509.876,Z 92.594,A -85,B 0,C 180,E1 -5563.172,E2 -5563.172} C_VEL
LIN {X 0,Y 509.866,Z 92.595,A -85,B 0,C 180,E1 -5565.632,E2 -5565.632} C_VEL
LIN {X 0,Y 509.922,Z 92.592,A -85,B 0,C 180,E1 -5568.872,E2 -5568.872} C_VEL
LIN {X 0,Y 509.918,Z 92.591,A -85,B 0,C 180,E1 -5572.076,E2 -5572.076} C_VEL
LIN {X 0,Y 509.972,Z 92.589,A -85,B 0,C 180,E1 -5574.462,E2 -5574.462} C_VEL
LIN {X 0,Y 510.057,Z 92.569,A -85,B 0,C 180,E1 -5577.628,E2 -5577.628} C_VEL
LIN {X 0,Y 510.046,Z 92.57,A -85,B 0,C 180,E1 -5580.787,E2 -5580.787} C_VEL
LIN {X 0,Y 509.932,Z 92.587,A -85,B 0,C 180,E1 -5583.158,E2 -5583.158} C_VEL
LIN {X 0,Y 509.941,Z 92.588,A -85,B 0,C 180,E1 -5586.327,E2 -5586.327} C_VEL
LIN {X 0,Y 509.907,Z 92.588,A -85,B 0,C 180,E1 -5588.717,E2 -5588.717} C_VEL
LIN {X 0,Y 509.906,Z 92.594,A -85,B 0,C 180,E1 -5591.929,E2 -5591.929} C_VEL
LIN {X 0,Y 509.894,Z 92.595,A -85,B 0,C 180,E1 -5595.239,E2 -5595.239} C_VEL
LIN {X 0,Y 509.855,Z 92.597,A -85,B 0,C 180,E1 -5598.481,E2 -5598.481} C_VEL
LIN {X 0,Y 509.842,Z 92.6,A -85,B 0,C 180,E1 -5600.998,E2 -5600.998} C_VEL
LIN {X 0,Y 509.814,Z 92.606,A -85,B 0,C 180,E1 -5603.561,E2 -5603.561} C_VEL
LIN {X 0,Y 509.873,Z 92.593,A -85,B 0,C 180,E1 -5606.368,E2 -5606.368} C_VEL
LIN {X 0,Y 509.863,Z 92.6,A -85,B 0,C 180,E1 -5608.841,E2 -5608.841} C_VEL
LIN {X 0,Y 509.807,Z 92.604,A -85,B 0,C 180,E1 -5611.587,E2 -5611.587} C_VEL
LIN {X 0,Y 509.825,Z 92.599,A -85,B 0,C 180,E1 -5614.411,E2 -5614.411} C_VEL
LIN {X 0,Y 509.8,Z 92.602,A -85,B 0,C 180,E1 -5617.337,E2 -5617.337} C_VEL
LIN {X 0,Y 509.821,Z 92.607,A -85,B 0,C 180,E1 -5620.379,E2 -5620.379} C_VEL
LIN {X 0,Y 509.804,Z 92.606,A -85,B 0,C 180,E1 -5623.059,E2 -5623.059} C_VEL
LIN {X 0,Y 509.801,Z 92.605,A -85,B 0,C 180,E1 -5625.79,E2 -5625.79} C_VEL
LIN {X 0,Y 509.823,Z 92.609,A -85,B 0,C 180,E1 -5628.57,E2 -5628.57} C_VEL
LIN {X 0,Y 509.848,Z 92.666,A -85,B 0,C 180,E1 -5630.902,E2 -5630.902} C_VEL
LIN {X 0,Y 511.523,Z 101.46,A -85,B 0,C 180,E1 -5632.556,E2 -5632.556} C_VEL
LIN {X 0,Y 511.44,Z 106.048,A -85,B 0,C 180,E1 -5633.361,E2 -5633.361} C_VEL
LIN {X 0,Y 510.92,Z 109.546,A -85,B 0,C 180,E1 -5633.875,E2 -5633.875} C_VEL
LIN {X 0,Y 509.521,Z 115.129,A -85,B 0,C 180,E1 -5634.456,E2 -5634.456} C_VEL
LIN {X 0,Y 508.004,Z 121.568,A -85,B 0,C 180,E1 -5634.901,E2 -5634.901} C_VEL
LIN {X 0,Y 507.207,Z 126.899,A -85,B 0,C 180,E1 -5635.127,E2 -5635.127} C_VEL
LIN {X 0,Y 507.025,Z 130.642,A -85,B 0,C 180,E1 -5635.214,E2 -5635.214} C_VEL
LIN {X 0,Y 506.155,Z 253.05,A -85,B 0,C 180,E1 -5637.005,E2 -5637.005} C_VEL
LIN {X 0,Y 505.881,Z 267.246,A -85,B 0,C 180,E1 -5637.369,E2 -5637.369} C_VEL
LIN {X 0,Y 505.523,Z 281.215,A -85,B 0,C 180,E1 -5637.898,E2 -5637.898} C_VEL
LIN {X 0,Y 505.102,Z 294.109,A -85,B 0,C 180,E1 -5638.547,E2 -5638.547} C_VEL
LIN {X 0,Y 504.65,Z 306.073,A -85,B 0,C 180,E1 -5639.31,E2 -5639.31} C_VEL
LIN {X 0,Y 504.181,Z 317.708,A -85,B 0,C 180,E1 -5640.224,E2 -5640.224} C_VEL
LIN {X 0,Y 503.7,Z 329.005,A -85,B 0,C 180,E1 -5641.307,E2 -5641.307} C_VEL
LIN {X 0,Y 503.235,Z 339.689,A -85,B 0,C 180,E1 -5642.556,E2 -5642.556} C_VEL
LIN {X 0,Y 502.861,Z 348.936,A -85,B 0,C 180,E1 -5643.879,E2 -5643.879} C_VEL
LIN {X 0,Y 502.6,Z 356.47,A -85,B 0,C 180,E1 -5645.196,E2 -5645.196} C_VEL
LIN {X 0,Y 502.382,Z 362.599,A -85,B 0,C 180,E1 -5646.502,E2 -5646.502} C_VEL
LIN {X 0,Y 502.266,Z 367.506,A -85,B 0,C 180,E1 -5647.801,E2 -5647.801} C_VEL
LIN {X 0,Y 502.197,Z 371.351,A -85,B 0,C 180,E1 -5649.091,E2 -5649.091} C_VEL
LIN {X 0,Y 502.084,Z 374.243,A -85,B 0,C 180,E1 -5650.369,E2 -5650.369} C_VEL
LIN {X 0,Y 502.012,Z 376.69,A -85,B 0,C 180,E1 -5652.061,E2 -5652.061} C_VEL
LIN {X 0,Y 501.98,Z 377.667,A -85,B 0,C 180,E1 -5653.738,E2 -5653.738} C_VEL
LIN {X 0,Y 502.034,Z 377.221,A -85,B 0,C 180,E1 -5655.404,E2 -5655.404} C_VEL
LIN {X 0,Y 502.05,Z 375.382,A -85,B 0,C 180,E1 -5657.056,E2 -5657.056} C_VEL
LIN {X 0,Y 502.163,Z 372.111,A -85,B 0,C 180,E1 -5658.699,E2 -5658.699} C_VEL
LIN {X 0,Y 502.212,Z 367.33,A -85,B 0,C 180,E1 -5660.331,E2 -5660.331} C_VEL
LIN {X 0,Y 502.366,Z 362.714,A -85,B 0,C 180,E1 -5661.552,E2 -5661.552} C_VEL
LIN {X 0,Y 502.624,Z 355.508,A -85,B 0,C 180,E1 -5663.065,E2 -5663.065} C_VEL
LIN {X 0,Y 502.874,Z 347.74,A -85,B 0,C 180,E1 -5664.385,E2 -5664.385} C_VEL
LIN {X 0,Y 503.249,Z 339.122,A -85,B 0,C 180,E1 -5665.594,E2 -5665.594} C_VEL
LIN {X 0,Y 503.697,Z 328.724,A -85,B 0,C 180,E1 -5666.799,E2 -5666.799} C_VEL
LIN {X 0,Y 504.149,Z 317.146,A -85,B 0,C 180,E1 -5667.902,E2 -5667.902} C_VEL
LIN {X 0,Y 504.606,Z 305.574,A -85,B 0,C 180,E1 -5668.802,E2 -5668.802} C_VEL
LIN {X 0,Y 505.144,Z 292.828,A -85,B 0,C 180,E1 -5669.6,E2 -5669.6} C_VEL
LIN {X 0,Y 505.567,Z 279.628,A -85,B 0,C 180,E1 -5670.248,E2 -5670.248} C_VEL
LIN {X 0,Y 505.881,Z 265.171,A -85,B 0,C 180,E1 -5670.77,E2 -5670.77} C_VEL
LIN {X 0,Y 506.07,Z 251.013,A -85,B 0,C 180,E1 -5671.109,E2 -5671.109} C_VEL
LIN {X 0,Y 506.936,Z 129.75,A -85,B 0,C 180,E1 -5672.87,E2 -5672.87} C_VEL
LIN {X 0,Y 504.132,Z 116.392,A -85,B 0,C 180,E1 -5673.195,E2 -5673.195} C_VEL
LIN {X 0,Y 504.637,Z 102.618,A -85,B 0,C 180,E1 -5675.593,E2 -5675.593} C_VEL
LIN {X 0,Y 502.927,Z 93.465,A -85,B 0,C 180,E1 -5677.306,E2 -5677.306} C_VEL
LIN {X 0,Y 502.805,Z 93.478,A -85,B 0,C 180,E1 -5680.468,E2 -5680.468} C_VEL
LIN {X 0,Y 502.828,Z 93.476,A -85,B 0,C 180,E1 -5682.921,E2 -5682.921} C_VEL
LIN {X 0,Y 502.845,Z 93.473,A -85,B 0,C 180,E1 -5685.399,E2 -5685.399} C_VEL
LIN {X 0,Y 502.826,Z 93.473,A -85,B 0,C 180,E1 -5688.129,E2 -5688.129} C_VEL
LIN {X 0,Y 502.77,Z 93.484,A -85,B 0,C 180,E1 -5691.31,E2 -5691.31} C_VEL
LIN {X 0,Y 502.789,Z 93.478,A -85,B 0,C 180,E1 -5693.912,E2 -5693.912} C_VEL
LIN {X 0,Y 502.843,Z 93.469,A -85,B 0,C 180,E1 -5696.566,E2 -5696.566} C_VEL
LIN {X 0,Y 502.805,Z 93.482,A -85,B 0,C 180,E1 -5699.288,E2 -5699.288} C_VEL
LIN {X 0,Y 502.762,Z 93.479,A -85,B 0,C 180,E1 -5702.085,E2 -5702.085} C_VEL
LIN {X 0,Y 502.797,Z 93.482,A -85,B 0,C 180,E1 -5704.964,E2 -5704.964} C_VEL
LIN {X 0,Y 502.772,Z 93.478,A -85,B 0,C 180,E1 -5707.954,E2 -5707.954} C_VEL
LIN {X 0,Y 502.801,Z 93.481,A -85,B 0,C 180,E1 -5710.999,E2 -5710.999} C_VEL
LIN {X 0,Y 502.776,Z 93.479,A -85,B 0,C 180,E1 -5713.381,E2 -5713.381} C_VEL
LIN {X 0,Y 502.804,Z 93.481,A -85,B 0,C 180,E1 -5716.62,E2 -5716.62} C_VEL
LIN {X 0,Y 502.801,Z 93.478,A -85,B 0,C 180,E1 -5719.005,E2 -5719.005} C_VEL
LIN {X 0,Y 502.772,Z 93.48,A -85,B 0,C 180,E1 -5722.049,E2 -5722.049} C_VEL
LIN {X 0,Y 502.785,Z 93.478,A -85,B 0,C 180,E1 -5725.038,E2 -5725.038} C_VEL
LIN {X 0,Y 502.765,Z 93.482,A -85,B 0,C 180,E1 -5727.918,E2 -5727.918} C_VEL
LIN {X 0,Y 502.814,Z 93.475,A -85,B 0,C 180,E1 -5730.716,E2 -5730.716} C_VEL
LIN {X 0,Y 502.857,Z 93.468,A -85,B 0,C 180,E1 -5733.437,E2 -5733.437} C_VEL
LIN {X 0,Y 502.8,Z 93.483,A -85,B 0,C 180,E1 -5736.09,E2 -5736.09} C_VEL
LIN {X 0,Y 502.781,Z 93.477,A -85,B 0,C 180,E1 -5738.692,E2 -5738.692} C_VEL
LIN {X 0,Y 502.827,Z 93.479,A -85,B 0,C 180,E1 -5741.88,E2 -5741.88} C_VEL
LIN {X 0,Y 502.821,Z 93.472,A -85,B 0,C 180,E1 -5744.665,E2 -5744.665} C_VEL
LIN {X 0,Y 502.883,Z 93.468,A -85,B 0,C 180,E1 -5748.029,E2 -5748.029} C_VEL
LIN {X 0,Y 502.865,Z 93.469,A -85,B 0,C 180,E1 -5751.16,E2 -5751.16} C_VEL
LIN {X 0,Y 502.916,Z 93.468,A -85,B 0,C 180,E1 -5753.584,E2 -5753.584} C_VEL
LIN {X 0,Y 502.893,Z 93.464,A -85,B 0,C 180,E1 -5756.798,E2 -5756.798} C_VEL
LIN {X 0,Y 503.026,Z 93.452,A -85,B 0,C 180,E1 -5759.202,E2 -5759.202} C_VEL
LIN {X 0,Y 502.894,Z 93.467,A -85,B 0,C 180,E1 -5761.604,E2 -5761.604} C_VEL
LIN {X 0,Y 502.894,Z 93.471,A -85,B 0,C 180,E1 -5763.207,E2 -5763.207} C_VEL
LIN {X 0,Y 502.92,Z 93.46,A -85,B 0,C 180,E1 -5766.421,E2 -5766.421} C_VEL
LIN {X 0,Y 502.867,Z 93.471,A -85,B 0,C 180,E1 -5768.846,E2 -5768.846} C_VEL
LIN {X 0,Y 502.839,Z 93.47,A -85,B 0,C 180,E1 -5772.104,E2 -5772.104} C_VEL
LIN {X 0,Y 502.842,Z 93.471,A -85,B 0,C 180,E1 -5775.402,E2 -5775.402} C_VEL
LIN {X 0,Y 502.841,Z 93.47,A -85,B 0,C 180,E1 -5778.125,E2 -5778.125} C_VEL
LIN {X 0,Y 502.824,Z 93.477,A -85,B 0,C 180,E1 -5780.538,E2 -5780.538} C_VEL
LIN {X 0,Y 502.793,Z 93.478,A -85,B 0,C 180,E1 -5783.043,E2 -5783.043} C_VEL
LIN {X 0,Y 502.838,Z 93.47,A -85,B 0,C 180,E1 -5785.678,E2 -5785.678} C_VEL
LIN {X 0,Y 502.837,Z 93.477,A -85,B 0,C 180,E1 -5788.375,E2 -5788.375} C_VEL
LIN {X 0,Y 502.79,Z 93.476,A -85,B 0,C 180,E1 -5791.501,E2 -5791.501} C_VEL
LIN {X 0,Y 502.802,Z 93.48,A -85,B 0,C 180,E1 -5794.446,E2 -5794.446} C_VEL
LIN {X 0,Y 502.778,Z 93.477,A -85,B 0,C 180,E1 -5797.18,E2 -5797.18} C_VEL
LIN {X 0,Y 502.786,Z 93.483,A -85,B 0,C 180,E1 -5800.017,E2 -5800.017} C_VEL
LIN {X 0,Y 502.802,Z 93.48,A -85,B 0,C 180,E1 -5802.201,E2 -5802.201} C_VEL
LIN {X 0,Y 502.8,Z 93.477,A -85,B 0,C 180,E1 -5805.47,E2 -5805.47} C_VEL
LIN {X 0,Y 502.82,Z 93.472,A -85,B 0,C 180,E1 -5808.936,E2 -5808.936} C_VEL
LIN {X 0,Y 502.793,Z 93.479,A -85,B 0,C 180,E1 -5812.048,E2 -5812.048} C_VEL
LIN {X 0,Y 502.799,Z 93.476,A -85,B 0,C 180,E1 -5815.036,E2 -5815.036} C_VEL
LIN {X 0,Y 502.783,Z 93.482,A -85,B 0,C 180,E1 -5817.917,E2 -5817.917} C_VEL
LIN {X 0,Y 502.824,Z 93.476,A -85,B 0,C 180,E1 -5820.714,E2 -5820.714} C_VEL
LIN {X 0,Y 502.865,Z 93.484,A -85,B 0,C 180,E1 -5823.441,E2 -5823.441} C_VEL
LIN {X 0,Y 505.219,Z 105.001,A -85,B 0,C 180,E1 -5825.336,E2 -5825.336} C_VEL
LIN {X 0,Y 504.802,Z 119.269,A -85,B 0,C 180,E1 -5827.49,E2 -5827.49} C_VEL
LIN {X 0,Y 504.162,Z 139.202,A -85,B 0,C 180,E1 -5830.456,E2 -5830.456} C_VEL
LIN {X 0,Y 504.066,Z 141.854,A -85,B 0,C 180,E1 -5830.847,E2 -5830.847} C_VEL
LIN {X 0,Y 506.898,Z 158.886,A -85,B 0,C 180,E1 -5831.209,E2 -5831.209} C_VEL
LIN {X 0,Y 505.975,Z 279.619,A -85,B 0,C 180,E1 -5832.964,E2 -5832.964} C_VEL
LIN {X 0,Y 505.679,Z 294.072,A -85,B 0,C 180,E1 -5833.334,E2 -5833.334} C_VEL
LIN {X 0,Y 505.336,Z 307.838,A -85,B 0,C 180,E1 -5833.851,E2 -5833.851} C_VEL
LIN {X 0,Y 504.835,Z 321.882,A -85,B 0,C 180,E1 -5834.56,E2 -5834.56} C_VEL
LIN {X 0,Y 504.327,Z 334.436,A -85,B 0,C 180,E1 -5835.371,E2 -5835.371} C_VEL
LIN {X 0,Y 503.775,Z 347.081,A -85,B 0,C 180,E1 -5836.385,E2 -5836.385} C_VEL
LIN {X 0,Y 503.394,Z 357.708,A -85,B 0,C 180,E1 -5837.432,E2 -5837.432} C_VEL
LIN {X 0,Y 502.983,Z 368.441,A -85,B 0,C 180,E1 -5838.72,E2 -5838.72} C_VEL
LIN {X 0,Y 502.66,Z 376.82,A -85,B 0,C 180,E1 -5839.936,E2 -5839.936} C_VEL
LIN {X 0,Y 502.41,Z 384.83,A -85,B 0,C 180,E1 -5841.352,E2 -5841.352} C_VEL
LIN {X 0,Y 502.253,Z 391.281,A -85,B 0,C 180,E1 -5842.766,E2 -5842.766} C_VEL
LIN {X 0,Y 502.174,Z 397,A -85,B 0,C 180,E1 -5844.379,E2 -5844.379} C_VEL
LIN {X 0,Y 502.112,Z 401.147,A -85,B 0,C 180,E1 -5845.988,E2 -5845.988} C_VEL
LIN {X 0,Y 502.091,Z 403.855,A -85,B 0,C 180,E1 -5847.594,E2 -5847.594} C_VEL
LIN {X 0,Y 501.989,Z 405.193,A -85,B 0,C 180,E1 -5849.199,E2 -5849.199} C_VEL
LIN {X 0,Y 501.989,Z 405.188,A -85,B 0,C 180,E1 -5850.803,E2 -5850.803} C_VEL
LIN {X 0,Y 502.091,Z 403.844,A -85,B 0,C 180,E1 -5852.408,E2 -5852.408} C_VEL
LIN {X 0,Y 502.113,Z 401.128,A -85,B 0,C 180,E1 -5854.014,E2 -5854.014} C_VEL
LIN {X 0,Y 502.177,Z 396.967,A -85,B 0,C 180,E1 -5855.623,E2 -5855.623} C_VEL
LIN {X 0,Y 502.255,Z 391.235,A -85,B 0,C 180,E1 -5857.236,E2 -5857.236} C_VEL
LIN {X 0,Y 502.412,Z 384.776,A -85,B 0,C 180,E1 -5858.65,E2 -5858.65} C_VEL
LIN {X 0,Y 502.662,Z 376.754,A -85,B 0,C 180,E1 -5860.066,E2 -5860.066} C_VEL
LIN {X 0,Y 502.987,Z 368.369,A -85,B 0,C 180,E1 -5861.282,E2 -5861.282} C_VEL
LIN {X 0,Y 503.36,Z 358.639,A -85,B 0,C 180,E1 -5862.459,E2 -5862.459} C_VEL
LIN {X 0,Y 503.755,Z 348.132,A -85,B 0,C 180,E1 -5863.515,E2 -5863.515} C_VEL
LIN {X 0,Y 504.244,Z 335.837,A -85,B 0,C 180,E1 -5864.531,E2 -5864.531} C_VEL
LIN {X 0,Y 504.745,Z 323.656,A -85,B 0,C 180,E1 -5865.341,E2 -5865.341} C_VEL
LIN {X 0,Y 505.27,Z 310.143,A -85,B 0,C 180,E1 -5866.049,E2 -5866.049} C_VEL
LIN {X 0,Y 505.645,Z 296.473,A -85,B 0,C 180,E1 -5866.592,E2 -5866.592} C_VEL
LIN {X 0,Y 505.954,Z 282.202,A -85,B 0,C 180,E1 -5866.987,E2 -5866.987} C_VEL
LIN {X 0,Y 506.236,Z 260.069,A -85,B 0,C 180,E1 -5867.341,E2 -5867.341} C_VEL
LIN {X 0,Y 506.913,Z 158.423,A -85,B 0,C 180,E1 -5868.811,E2 -5868.811} C_VEL
LIN {X 0,Y 504.067,Z 141.619,A -85,B 0,C 180,E1 -5869.192,E2 -5869.192} C_VEL
LIN {X 0,Y 504.751,Z 122.289,A -85,B 0,C 180,E1 -5872.083,E2 -5872.083} C_VEL
LIN {X 0,Y 505.337,Z 105.396,A -85,B 0,C 180,E1 -5874.661,E2 -5874.661} C_VEL
LIN {X 0,Y 502.847,Z 93.476,A -85,B 0,C 180,E1 -5876.694,E2 -5876.694} C_VEL
LIN {X 0,Y 502.834,Z 93.475,A -85,B 0,C 180,E1 -5879.288,E2 -5879.288} C_VEL
LIN {X 0,Y 502.793,Z 93.484,A -85,B 0,C 180,E1 -5882.085,E2 -5882.085} C_VEL
LIN {X 0,Y 502.805,Z 93.477,A -85,B 0,C 180,E1 -5884.966,E2 -5884.966} C_VEL
LIN {X 0,Y 502.804,Z 93.48,A -85,B 0,C 180,E1 -5888.486,E2 -5888.486} C_VEL
LIN {X 0,Y 502.812,Z 93.472,A -85,B 0,C 180,E1 -5891.068,E2 -5891.068} C_VEL
LIN {X 0,Y 502.791,Z 93.479,A -85,B 0,C 180,E1 -5894.34,E2 -5894.34} C_VEL
LIN {X 0,Y 502.784,Z 93.478,A -85,B 0,C 180,E1 -5896.768,E2 -5896.768} C_VEL
LIN {X 0,Y 502.812,Z 93.466,A -85,B 0,C 180,E1 -5899.007,E2 -5899.007} C_VEL
LIN {X 0,Y 502.802,Z 93.476,A -85,B 0,C 180,E1 -5902.045,E2 -5902.045} C_VEL
LIN {X 0,Y 502.807,Z 93.477,A -85,B 0,C 180,E1 -5905.033,E2 -5905.033} C_VEL
LIN {X 0,Y 502.795,Z 93.477,A -85,B 0,C 180,E1 -5907.914,E2 -5907.914} C_VEL
LIN {X 0,Y 502.825,Z 93.474,A -85,B 0,C 180,E1 -5910.71,E2 -5910.71} C_VEL
LIN {X 0,Y 502.857,Z 93.473,A -85,B 0,C 180,E1 -5913.443,E2 -5913.443} C_VEL
LIN {X 0,Y 502.786,Z 93.473,A -85,B 0,C 180,E1 -5916.084,E2 -5916.084} C_VEL
LIN {X 0,Y 502.794,Z 93.481,A -85,B 0,C 180,E1 -5918.687,E2 -5918.687} C_VEL
LIN {X 0,Y 502.835,Z 93.474,A -85,B 0,C 180,E1 -5921.246,E2 -5921.246} C_VEL
LIN {X 0,Y 502.861,Z 93.47,A -85,B 0,C 180,E1 -5924.599,E2 -5924.599} C_VEL
LIN {X 0,Y 502.888,Z 93.464,A -85,B 0,C 180,E1 -5928.037,E2 -5928.037} C_VEL
LIN {X 0,Y 502.872,Z 93.466,A -85,B 0,C 180,E1 -5931.154,E2 -5931.154} C_VEL
LIN {X 0,Y 502.925,Z 93.467,A -85,B 0,C 180,E1 -5934.384,E2 -5934.384} C_VEL
LIN {X 0,Y 503.026,Z 93.445,A -85,B 0,C 180,E1 -5937.595,E2 -5937.595} C_VEL
LIN {X 0,Y 502.997,Z 93.448,A -85,B 0,C 180,E1 -5940.798,E2 -5940.798} C_VEL
LIN {X 0,Y 503.024,Z 93.451,A -85,B 0,C 180,E1 -5942.4,E2 -5942.4} C_VEL
LIN {X 0,Y 502.929,Z 93.461,A -85,B 0,C 180,E1 -5945.611,E2 -5945.611} C_VEL
LIN {X 0,Y 502.867,Z 93.465,A -85,B 0,C 180,E1 -5948.84,E2 -5948.84} C_VEL
LIN {X 0,Y 502.847,Z 93.471,A -85,B 0,C 180,E1 -5952.099,E2 -5952.099} C_VEL
LIN {X 0,Y 502.848,Z 93.475,A -85,B 0,C 180,E1 -5955.396,E2 -5955.396} C_VEL
LIN {X 0,Y 502.82,Z 93.474,A -85,B 0,C 180,E1 -5958.749,E2 -5958.749} C_VEL
LIN {X 0,Y 502.777,Z 93.484,A -85,B 0,C 180,E1 -5961.308,E2 -5961.308} C_VEL
LIN {X 0,Y 502.764,Z 93.481,A -85,B 0,C 180,E1 -5963.911,E2 -5963.911} C_VEL
LIN {X 0,Y 502.829,Z 93.471,A -85,B 0,C 180,E1 -5966.564,E2 -5966.564} C_VEL
LIN {X 0,Y 502.813,Z 93.471,A -85,B 0,C 180,E1 -5969.284,E2 -5969.284} C_VEL
LIN {X 0,Y 502.771,Z 93.48,A -85,B 0,C 180,E1 -5972.081,E2 -5972.081} C_VEL
LIN {X 0,Y 502.782,Z 93.482,A -85,B 0,C 180,E1 -5974.963,E2 -5974.963} C_VEL
LIN {X 0,Y 502.776,Z 93.476,A -85,B 0,C 180,E1 -5977.951,E2 -5977.951} C_VEL
LIN {X 0,Y 502.803,Z 93.478,A -85,B 0,C 180,E1 -5981.062,E2 -5981.062} C_VEL
LIN {X 0,Y 502.766,Z 93.487,A -85,B 0,C 180,E1 -5984.526,E2 -5984.526} C_VEL
LIN {X 0,Y 502.773,Z 93.485,A -85,B 0,C 180,E1 -5987.857,E2 -5987.857} C_VEL
LIN {X 0,Y 502.793,Z 93.549,A -85,B 0,C 180,E1 -5990.667,E2 -5990.667} C_VEL
LIN {X 0,Y 504.637,Z 103.324,A -85,B 0,C 180,E1 -5992.538,E2 -5992.538} C_VEL
LIN {X 0,Y 504.217,Z 116.735,A -85,B 0,C 180,E1 -5994.891,E2 -5994.891} C_VEL
LIN {X 0,Y 507.025,Z 130.642,A -85,B 0,C 180,E1 -5995.214,E2 -5995.214} C_VEL
LIN {X 0,Y 506.384,Z 136.493,A -85,B 0,C 180,E1 -5995.274,E2 -5995.274} C_VEL
LIN {X 0,Y 500.803,Z 155.542,A -85,B 0,C 180,E1 -5995.33,E2 -5995.33} C_VEL
LIN {X 0,Y 500.162,Z 161.393,A -85,B 0,C 180,E1 -5995.392,E2 -5995.392} C_VEL
LIN {X 0,Y 499.389,Z 253.831,A -85,B 0,C 180,E1 -5996.771,E2 -5996.771} C_VEL
LIN {X 0,Y 499.113,Z 267.806,A -85,B 0,C 180,E1 -5997.141,E2 -5997.141} C_VEL
LIN {X 0,Y 498.718,Z 281.672,A -85,B 0,C 180,E1 -5997.676,E2 -5997.676} C_VEL
LIN {X 0,Y 498.283,Z 294.012,A -85,B 0,C 180,E1 -5998.307,E2 -5998.307} C_VEL
LIN {X 0,Y 497.803,Z 306.274,A -85,B 0,C 180,E1 -5999.099,E2 -5999.099} C_VEL
LIN {X 0,Y 497.23,Z 318.933,A -85,B 0,C 180,E1 -6000.116,E2 -6000.116} C_VEL
LIN {X 0,Y 496.722,Z 330.345,A -85,B 0,C 180,E1 -6001.244,E2 -6001.244} C_VEL
LIN {X 0,Y 496.253,Z 339.707,A -85,B 0,C 180,E1 -6002.366,E2 -6002.366} C_VEL
LIN {X 0,Y 495.846,Z 349.076,A -85,B 0,C 180,E1 -6003.721,E2 -6003.721} C_VEL
LIN {X 0,Y 495.543,Z 357.201,A -85,B 0,C 180,E1 -6005.175,E2 -6005.175} C_VEL
LIN {X 0,Y 495.304,Z 363.585,A -85,B 0,C 180,E1 -6006.589,E2 -6006.589} C_VEL
LIN {X 0,Y 495.194,Z 368.366,A -85,B 0,C 180,E1 -6007.907,E2 -6007.907} C_VEL
LIN {X 0,Y 495.089,Z 372.792,A -85,B 0,C 180,E1 -6009.524,E2 -6009.524} C_VEL
LIN {X 0,Y 494.953,Z 375.526,A -85,B 0,C 180,E1 -6010.937,E2 -6010.937} C_VEL
LIN {X 0,Y 494.903,Z 377.417,A -85,B 0,C 180,E1 -6012.648,E2 -6012.648} C_VEL
LIN {X 0,Y 494.874,Z 377.863,A -85,B 0,C 180,E1 -6014.345,E2 -6014.345} C_VEL
LIN {X 0,Y 494.926,Z 376.898,A -85,B 0,C 180,E1 -6016.03,E2 -6016.03} C_VEL
LIN {X 0,Y 494.995,Z 374.537,A -85,B 0,C 180,E1 -6017.702,E2 -6017.702} C_VEL
LIN {X 0,Y 495.105,Z 370.746,A -85,B 0,C 180,E1 -6019.365,E2 -6019.365} C_VEL
LIN {X 0,Y 495.17,Z 366.876,A -85,B 0,C 180,E1 -6020.605,E2 -6020.605} C_VEL
LIN {X 0,Y 495.33,Z 362.1,A -85,B 0,C 180,E1 -6021.842,E2 -6021.842} C_VEL
LIN {X 0,Y 495.61,Z 355.333,A -85,B 0,C 180,E1 -6023.257,E2 -6023.257} C_VEL
LIN {X 0,Y 495.9,Z 346.71,A -85,B 0,C 180,E1 -6024.713,E2 -6024.713} C_VEL
LIN {X 0,Y 496.301,Z 337.854,A -85,B 0,C 180,E1 -6025.939,E2 -6025.939} C_VEL
LIN {X 0,Y 496.805,Z 327.166,A -85,B 0,C 180,E1 -6027.161,E2 -6027.161} C_VEL
LIN {X 0,Y 497.313,Z 316.367,A -85,B 0,C 180,E1 -6028.177,E2 -6028.177} C_VEL
LIN {X 0,Y 497.795,Z 304.593,A -85,B 0,C 180,E1 -6029.089,E2 -6029.089} C_VEL
LIN {X 0,Y 498.355,Z 291.545,A -85,B 0,C 180,E1 -6029.898,E2 -6029.898} C_VEL
LIN {X 0,Y 498.755,Z 279.062,A -85,B 0,C 180,E1 -6030.503,E2 -6030.503} C_VEL
LIN {X 0,Y 499.087,Z 265.344,A -85,B 0,C 180,E1 -6030.999,E2 -6030.999} C_VEL
LIN {X 0,Y 499.28,Z 251.339,A -85,B 0,C 180,E1 -6031.34,E2 -6031.34} C_VEL
LIN {X 0,Y 500.169,Z 130.462,A -85,B 0,C 180,E1 -6033.118,E2 -6033.118} C_VEL
LIN {X 0,Y 497.225,Z 116.673,A -85,B 0,C 180,E1 -6033.443,E2 -6033.443} C_VEL
LIN {X 0,Y 497.711,Z 104.022,A -85,B 0,C 180,E1 -6035.671,E2 -6035.671} C_VEL
LIN {X 0,Y 495.878,Z 94.344,A -85,B 0,C 180,E1 -6037.511,E2 -6037.511} C_VEL
LIN {X 0,Y 495.763,Z 94.355,A -85,B 0,C 180,E1 -6040.618,E2 -6040.618} C_VEL
LIN {X 0,Y 495.777,Z 94.356,A -85,B 0,C 180,E1 -6043.108,E2 -6043.108} C_VEL
LIN {X 0,Y 495.787,Z 94.356,A -85,B 0,C 180,E1 -6045.623,E2 -6045.623} C_VEL
LIN {X 0,Y 495.792,Z 94.348,A -85,B 0,C 180,E1 -6048.256,E2 -6048.256} C_VEL
LIN {X 0,Y 495.734,Z 94.361,A -85,B 0,C 180,E1 -6051.628,E2 -6051.628} C_VEL
LIN {X 0,Y 495.771,Z 94.352,A -85,B 0,C 180,E1 -6054.882,E2 -6054.882} C_VEL
LIN {X 0,Y 495.75,Z 94.354,A -85,B 0,C 180,E1 -6057.892,E2 -6057.892} C_VEL
LIN {X 0,Y 495.729,Z 94.357,A -85,B 0,C 180,E1 -6060.687,E2 -6060.687} C_VEL
LIN {X 0,Y 495.731,Z 94.357,A -85,B 0,C 180,E1 -6063.565,E2 -6063.565} C_VEL
LIN {X 0,Y 495.716,Z 94.359,A -85,B 0,C 180,E1 -6066.543,E2 -6066.543} C_VEL
LIN {X 0,Y 495.777,Z 94.35,A -85,B 0,C 180,E1 -6069.634,E2 -6069.634} C_VEL
LIN {X 0,Y 495.744,Z 94.361,A -85,B 0,C 180,E1 -6072.879,E2 -6072.879} C_VEL
LIN {X 0,Y 495.763,Z 94.354,A -85,B 0,C 180,E1 -6076.299,E2 -6076.299} C_VEL
LIN {X 0,Y 495.758,Z 94.352,A -85,B 0,C 180,E1 -6079.304,E2 -6079.304} C_VEL
LIN {X 0,Y 495.74,Z 94.354,A -85,B 0,C 180,E1 -6081.412,E2 -6081.412} C_VEL
LIN {X 0,Y 495.733,Z 94.363,A -85,B 0,C 180,E1 -6084.466,E2 -6084.466} C_VEL
LIN {X 0,Y 495.744,Z 94.353,A -85,B 0,C 180,E1 -6087.408,E2 -6087.408} C_VEL
LIN {X 0,Y 495.757,Z 94.36,A -85,B 0,C 180,E1 -6090.257,E2 -6090.257} C_VEL
LIN {X 0,Y 495.81,Z 94.345,A -85,B 0,C 180,E1 -6093.251,E2 -6093.251} C_VEL
LIN {X 0,Y 495.752,Z 94.356,A -85,B 0,C 180,E1 -6095.729,E2 -6095.729} C_VEL
LIN {X 0,Y 495.746,Z 94.357,A -85,B 0,C 180,E1 -6098.375,E2 -6098.375} C_VEL
LIN {X 0,Y 495.766,Z 94.351,A -85,B 0,C 180,E1 -6100.974,E2 -6100.974} C_VEL
LIN {X 0,Y 495.764,Z 94.355,A -85,B 0,C 180,E1 -6103.533,E2 -6103.533} C_VEL
LIN {X 0,Y 495.778,Z 94.354,A -85,B 0,C 180,E1 -6106.058,E2 -6106.058} C_VEL
LIN {X 0,Y 495.854,Z 94.34,A -85,B 0,C 180,E1 -6108.558,E2 -6108.558} C_VEL
LIN {X 0,Y 495.86,Z 94.344,A -85,B 0,C 180,E1 -6111.855,E2 -6111.855} C_VEL
LIN {X 0,Y 495.893,Z 94.335,A -85,B 0,C 180,E1 -6114.309,E2 -6114.309} C_VEL
LIN {X 0,Y 495.983,Z 94.33,A -85,B 0,C 180,E1 -6117.566,E2 -6117.566} C_VEL
LIN {X 0,Y 495.987,Z 94.324,A -85,B 0,C 180,E1 -6120.003,E2 -6120.003} C_VEL
LIN {X 0,Y 495.984,Z 94.324,A -85,B 0,C 180,E1 -6122.439,E2 -6122.439} C_VEL
LIN {X 0,Y 495.888,Z 94.337,A -85,B 0,C 180,E1 -6125.696,E2 -6125.696} C_VEL
LIN {X 0,Y 495.865,Z 94.338,A -85,B 0,C 180,E1 -6128.15,E2 -6128.15} C_VEL
LIN {X 0,Y 495.844,Z 94.343,A -85,B 0,C 180,E1 -6131.448,E2 -6131.448} C_VEL
LIN {X 0,Y 495.783,Z 94.355,A -85,B 0,C 180,E1 -6134.785,E2 -6134.785} C_VEL
LIN {X 0,Y 495.781,Z 94.351,A -85,B 0,C 180,E1 -6137.321,E2 -6137.321} C_VEL
LIN {X 0,Y 495.766,Z 94.351,A -85,B 0,C 180,E1 -6139.893,E2 -6139.893} C_VEL
LIN {X 0,Y 495.754,Z 94.357,A -85,B 0,C 180,E1 -6142.863,E2 -6142.863} C_VEL
LIN {X 0,Y 495.796,Z 94.349,A -85,B 0,C 180,E1 -6146.07,E2 -6146.07} C_VEL
LIN {X 0,Y 495.769,Z 94.354,A -85,B 0,C 180,E1 -6148.817,E2 -6148.817} C_VEL
LIN {X 0,Y 495.753,Z 94.353,A -85,B 0,C 180,E1 -6151.727,E2 -6151.727} C_VEL
LIN {X 0,Y 495.772,Z 94.353,A -85,B 0,C 180,E1 -6154.697,E2 -6154.697} C_VEL
LIN {X 0,Y 495.728,Z 94.356,A -85,B 0,C 180,E1 -6157.564,E2 -6157.564} C_VEL
LIN {X 0,Y 495.765,Z 94.352,A -85,B 0,C 180,E1 -6160.702,E2 -6160.702} C_VEL
LIN {X 0,Y 495.733,Z 94.363,A -85,B 0,C 180,E1 -6164.003,E2 -6164.003} C_VEL
LIN {X 0,Y 495.724,Z 94.356,A -85,B 0,C 180,E1 -6167.119,E2 -6167.119} C_VEL
LIN {X 0,Y 495.758,Z 94.358,A -85,B 0,C 180,E1 -6169.955,E2 -6169.955} C_VEL
LIN {X 0,Y 495.727,Z 94.356,A -85,B 0,C 180,E1 -6172.555,E2 -6172.555} C_VEL
LIN {X 0,Y 495.778,Z 94.355,A -85,B 0,C 180,E1 -6175.458,E2 -6175.458} C_VEL
LIN {X 0,Y 495.755,Z 94.355,A -85,B 0,C 180,E1 -6178.365,E2 -6178.365} C_VEL
LIN {X 0,Y 495.788,Z 94.356,A -85,B 0,C 180,E1 -6181.509,E2 -6181.509} C_VEL
LIN {X 0,Y 495.831,Z 94.543,A -85,B 0,C 180,E1 -6183.251,E2 -6183.251} C_VEL
LIN {X 0,Y 498.258,Z 106.145,A -85,B 0,C 180,E1 -6185.19,E2 -6185.19} C_VEL
LIN {X 0,Y 498.09,Z 114.746,A -85,B 0,C 180,E1 -6186.514,E2 -6186.514} C_VEL
LIN {X 0,Y 497.366,Z 134.669,A -85,B 0,C 180,E1 -6189.531,E2 -6189.531} C_VEL
LIN {X 0,Y 497.124,Z 141.711,A -85,B 0,C 180,E1 -6190.584,E2 -6190.584} C_VEL
LIN {X 0,Y 500.148,Z 159.562,A -85,B 0,C 180,E1 -6190.967,E2 -6190.967} C_VEL
LIN {X 0,Y 499.199,Z 279.148,A -85,B 0,C 180,E1 -6192.726,E2 -6192.726} C_VEL
LIN {X 0,Y 498.873,Z 293.246,A -85,B 0,C 180,E1 -6193.083,E2 -6193.083} C_VEL
LIN {X 0,Y 498.517,Z 306.503,A -85,B 0,C 180,E1 -6193.577,E2 -6193.577} C_VEL
LIN {X 0,Y 498.004,Z 319.82,A -85,B 0,C 180,E1 -6194.238,E2 -6194.238} C_VEL
LIN {X 0,Y 497.499,Z 332.734,A -85,B 0,C 180,E1 -6195.061,E2 -6195.061} C_VEL
LIN {X 0,Y 496.91,Z 344.464,A -85,B 0,C 180,E1 -6195.985,E2 -6195.985} C_VEL
LIN {X 0,Y 496.425,Z 356.189,A -85,B 0,C 180,E1 -6197.117,E2 -6197.117} C_VEL
LIN {X 0,Y 496.006,Z 366.881,A -85,B 0,C 180,E1 -6198.379,E2 -6198.379} C_VEL
LIN {X 0,Y 495.682,Z 375.324,A -85,B 0,C 180,E1 -6199.586,E2 -6199.586} C_VEL
LIN {X 0,Y 495.385,Z 383.608,A -85,B 0,C 180,E1 -6201.023,E2 -6201.023} C_VEL
LIN {X 0,Y 495.207,Z 389.399,A -85,B 0,C 180,E1 -6202.253,E2 -6202.253} C_VEL
LIN {X 0,Y 495.107,Z 394.364,A -85,B 0,C 180,E1 -6203.542,E2 -6203.542} C_VEL
LIN {X 0,Y 495.028,Z 399.064,A -85,B 0,C 180,E1 -6205.115,E2 -6205.115} C_VEL
LIN {X 0,Y 495.034,Z 402.481,A -85,B 0,C 180,E1 -6206.746,E2 -6206.746} C_VEL
LIN {X 0,Y 494.961,Z 404.499,A -85,B 0,C 180,E1 -6208.374,E2 -6208.374} C_VEL
LIN {X 0,Y 494.901,Z 405.163,A -85,B 0,C 180,E1 -6210.001,E2 -6210.001} C_VEL
LIN {X 0,Y 494.961,Z 404.489,A -85,B 0,C 180,E1 -6211.628,E2 -6211.628} C_VEL
LIN {X 0,Y 495.035,Z 402.464,A -85,B 0,C 180,E1 -6213.257,E2 -6213.257} C_VEL
LIN {X 0,Y 495.029,Z 399.035,A -85,B 0,C 180,E1 -6214.888,E2 -6214.888} C_VEL
LIN {X 0,Y 495.111,Z 394.108,A -85,B 0,C 180,E1 -6216.522,E2 -6216.522} C_VEL
LIN {X 0,Y 495.276,Z 387.536,A -85,B 0,C 180,E1 -6218.159,E2 -6218.159} C_VEL
LIN {X 0,Y 495.505,Z 380.227,A -85,B 0,C 180,E1 -6219.595,E2 -6219.595} C_VEL
LIN {X 0,Y 495.864,Z 371.177,A -85,B 0,C 180,E1 -6221.032,E2 -6221.032} C_VEL
LIN {X 0,Y 496.225,Z 361.684,A -85,B 0,C 180,E1 -6222.267,E2 -6222.267} C_VEL
LIN {X 0,Y 496.666,Z 351.181,A -85,B 0,C 180,E1 -6223.399,E2 -6223.399} C_VEL
LIN {X 0,Y 497.165,Z 339.597,A -85,B 0,C 180,E1 -6224.428,E2 -6224.428} C_VEL
LIN {X 0,Y 497.751,Z 326.753,A -85,B 0,C 180,E1 -6225.353,E2 -6225.353} C_VEL
LIN {X 0,Y 498.281,Z 314.222,A -85,B 0,C 180,E1 -6226.07,E2 -6226.07} C_VEL
LIN {X 0,Y 498.672,Z 301.095,A -85,B 0,C 180,E1 -6226.657,E2 -6226.657} C_VEL
LIN {X 0,Y 499.072,Z 286.9,A -85,B 0,C 180,E1 -6227.115,E2 -6227.115} C_VEL
LIN {X 0,Y 499.35,Z 272.773,A -85,B 0,C 180,E1 -6227.403,E2 -6227.403} C_VEL
LIN {X 0,Y 500.206,Z 158.965,A -85,B 0,C 180,E1 -6229.073,E2 -6229.073} C_VEL
LIN {X 0,Y 497.181,Z 141.37,A -85,B 0,C 180,E1 -6229.488,E2 -6229.488} C_VEL
LIN {X 0,Y 498.001,Z 119.398,A -85,B 0,C 180,E1 -6232.837,E2 -6232.837} C_VEL
LIN {X 0,Y 498.457,Z 106.759,A -85,B 0,C 180,E1 -6234.802,E2 -6234.802} C_VEL
LIN {X 0,Y 495.825,Z 94.35,A -85,B 0,C 180,E1 -6236.975,E2 -6236.975} C_VEL
LIN {X 0,Y 495.775,Z 94.357,A -85,B 0,C 180,E1 -6240.147,E2 -6240.147} C_VEL
LIN {X 0,Y 495.801,Z 94.352,A -85,B 0,C 180,E1 -6243.244,E2 -6243.244} C_VEL
LIN {X 0,Y 495.724,Z 94.365,A -85,B 0,C 180,E1 -6246.087,E2 -6246.087} C_VEL
LIN {X 0,Y 495.772,Z 94.353,A -85,B 0,C 180,E1 -6248.768,E2 -6248.768} C_VEL
LIN {X 0,Y 495.763,Z 94.355,A -85,B 0,C 180,E1 -6251.782,E2 -6251.782} C_VEL
LIN {X 0,Y 495.75,Z 94.354,A -85,B 0,C 180,E1 -6255.141,E2 -6255.141} C_VEL
LIN {X 0,Y 495.764,Z 94.346,A -85,B 0,C 180,E1 -6258.218,E2 -6258.218} C_VEL
LIN {X 0,Y 495.759,Z 94.357,A -85,B 0,C 180,E1 -6261.407,E2 -6261.407} C_VEL
LIN {X 0,Y 495.757,Z 94.353,A -85,B 0,C 180,E1 -6264.461,E2 -6264.461} C_VEL
LIN {X 0,Y 495.779,Z 94.357,A -85,B 0,C 180,E1 -6267.405,E2 -6267.405} C_VEL
LIN {X 0,Y 495.775,Z 94.35,A -85,B 0,C 180,E1 -6270.252,E2 -6270.252} C_VEL
LIN {X 0,Y 495.787,Z 94.355,A -85,B 0,C 180,E1 -6273.261,E2 -6273.261} C_VEL
LIN {X 0,Y 495.754,Z 94.352,A -85,B 0,C 180,E1 -6276.611,E2 -6276.611} C_VEL
LIN {X 0,Y 495.792,Z 94.347,A -85,B 0,C 180,E1 -6279.323,E2 -6279.323} C_VEL
LIN {X 0,Y 495.791,Z 94.348,A -85,B 0,C 180,E1 -6281.827,E2 -6281.827} C_VEL
LIN {X 0,Y 495.836,Z 94.344,A -85,B 0,C 180,E1 -6284.547,E2 -6284.547} C_VEL
LIN {X 0,Y 495.84,Z 94.341,A -85,B 0,C 180,E1 -6287.963,E2 -6287.963} C_VEL
LIN {X 0,Y 495.842,Z 94.343,A -85,B 0,C 180,E1 -6291.028,E2 -6291.028} C_VEL
LIN {X 0,Y 495.88,Z 94.343,A -85,B 0,C 180,E1 -6294.304,E2 -6294.304} C_VEL
LIN {X 0,Y 495.994,Z 94.321,A -85,B 0,C 180,E1 -6297.561,E2 -6297.561} C_VEL
LIN {X 0,Y 495.949,Z 94.325,A -85,B 0,C 180,E1 -6300.809,E2 -6300.809} C_VEL
LIN {X 0,Y 495.992,Z 94.327,A -85,B 0,C 180,E1 -6302.434,E2 -6302.434} C_VEL
LIN {X 0,Y 495.885,Z 94.338,A -85,B 0,C 180,E1 -6305.691,E2 -6305.691} C_VEL
LIN {X 0,Y 495.837,Z 94.341,A -85,B 0,C 180,E1 -6308.967,E2 -6308.967} C_VEL
LIN {X 0,Y 495.83,Z 94.345,A -85,B 0,C 180,E1 -6312.031,E2 -6312.031} C_VEL
LIN {X 0,Y 495.824,Z 94.351,A -85,B 0,C 180,E1 -6315.448,E2 -6315.448} C_VEL
LIN {X 0,Y 495.776,Z 94.354,A -85,B 0,C 180,E1 -6319.025,E2 -6319.025} C_VEL
LIN {X 0,Y 495.737,Z 94.359,A -85,B 0,C 180,E1 -6321.626,E2 -6321.626} C_VEL
LIN {X 0,Y 495.71,Z 94.359,A -85,B 0,C 180,E1 -6324.273,E2 -6324.273} C_VEL
LIN {X 0,Y 495.775,Z 94.355,A -85,B 0,C 180,E1 -6326.972,E2 -6326.972} C_VEL
LIN {X 0,Y 495.756,Z 94.346,A -85,B 0,C 180,E1 -6329.743,E2 -6329.743} C_VEL
LIN {X 0,Y 495.754,Z 94.358,A -85,B 0,C 180,E1 -6332.591,E2 -6332.591} C_VEL
LIN {X 0,Y 495.733,Z 94.358,A -85,B 0,C 180,E1 -6335.534,E2 -6335.534} C_VEL
LIN {X 0,Y 495.742,Z 94.36,A -85,B 0,C 180,E1 -6338.764,E2 -6338.764} C_VEL
LIN {X 0,Y 495.739,Z 94.356,A -85,B 0,C 180,E1 -6341.778,E2 -6341.778} C_VEL
LIN {X 0,Y 495.717,Z 94.359,A -85,B 0,C 180,E1 -6345.137,E2 -6345.137} C_VEL
LIN {X 0,Y 495.728,Z 94.368,A -85,B 0,C 180,E1 -6348.215,E2 -6348.215} C_VEL
LIN {X 0,Y 495.735,Z 94.408,A -85,B 0,C 180,E1 -6350.416,E2 -6350.416} C_VEL
LIN {X 0,Y 497.62,Z 103.865,A -85,B 0,C 180,E1 -6352.263,E2 -6352.263} C_VEL
LIN {X 0,Y 497.55,Z 111.344,A -85,B 0,C 180,E1 -6353.616,E2 -6353.616} C_VEL
LIN {X 0,Y 497.351,Z 116.823,A -85,B 0,C 180,E1 -6354.593,E2 -6354.593} C_VEL
LIN {X 0,Y 500.354,Z 131.004,A -85,B 0,C 180,E1 -6354.943,E2 -6354.943} C_VEL
LIN {X 0,Y 500.162,Z 161.393,A -85,B 0,C 180,E1 -6355.392,E2 -6355.392} C_VEL
LIN {X 0,Y 499.54,Z 167.237,A -85,B 0,C 180,E1 -6355.454,E2 -6355.454} C_VEL
LIN {X 0,Y 493.955,Z 186.275,A -85,B 0,C 180,E1 -6355.514,E2 -6355.514} C_VEL
LIN {X 0,Y 493.167,Z 192.127,A -85,B 0,C 180,E1 -6355.57,E2 -6355.57} C_VEL
LIN {X 0,Y 492.661,Z 253.428,A -85,B 0,C 180,E1 -6356.502,E2 -6356.502} C_VEL
LIN {X 0,Y 492.364,Z 268.039,A -85,B 0,C 180,E1 -6356.892,E2 -6356.892} C_VEL
LIN {X 0,Y 491.946,Z 281.961,A -85,B 0,C 180,E1 -6357.437,E2 -6357.437} C_VEL
LIN {X 0,Y 491.403,Z 295.878,A -85,B 0,C 180,E1 -6358.17,E2 -6358.17} C_VEL
LIN {X 0,Y 490.824,Z 309.059,A -85,B 0,C 180,E1 -6359.064,E2 -6359.064} C_VEL
LIN {X 0,Y 490.306,Z 320.249,A -85,B 0,C 180,E1 -6360.006,E2 -6360.006} C_VEL
LIN {X 0,Y 489.758,Z 331.595,A -85,B 0,C 180,E1 -6361.17,E2 -6361.17} C_VEL
LIN {X 0,Y 489.224,Z 341.442,A -85,B 0,C 180,E1 -6362.399,E2 -6362.399} C_VEL
LIN {X 0,Y 488.794,Z 350.402,A -85,B 0,C 180,E1 -6363.759,E2 -6363.759} C_VEL
LIN {X 0,Y 488.507,Z 357.178,A -85,B 0,C 180,E1 -6364.997,E2 -6364.997} C_VEL
LIN {X 0,Y 488.269,Z 362.805,A -85,B 0,C 180,E1 -6366.232,E2 -6366.232} C_VEL
LIN {X 0,Y 488.162,Z 367.754,A -85,B 0,C 180,E1 -6367.571,E2 -6367.571} C_VEL
LIN {X 0,Y 488.045,Z 371.634,A -85,B 0,C 180,E1 -6368.898,E2 -6368.898} C_VEL
LIN {X 0,Y 487.96,Z 373.68,A -85,B 0,C 180,E1 -6369.776,E2 -6369.776} C_VEL
LIN {X 0,Y 487.834,Z 376.576,A -85,B 0,C 180,E1 -6371.521,E2 -6371.521} C_VEL
LIN {X 0,Y 487.783,Z 377.965,A -85,B 0,C 180,E1 -6373.251,E2 -6373.251} C_VEL
LIN {X 0,Y 487.833,Z 377.884,A -85,B 0,C 180,E1 -6374.969,E2 -6374.969} C_VEL
LIN {X 0,Y 487.862,Z 376.4,A -85,B 0,C 180,E1 -6376.673,E2 -6376.673} C_VEL
LIN {X 0,Y 487.977,Z 373.509,A -85,B 0,C 180,E1 -6378.366,E2 -6378.366} C_VEL
LIN {X 0,Y 488.053,Z 369.167,A -85,B 0,C 180,E1 -6380.048,E2 -6380.048} C_VEL
LIN {X 0,Y 488.261,Z 363.25,A -85,B 0,C 180,E1 -6381.723,E2 -6381.723} C_VEL
LIN {X 0,Y 488.487,Z 357.274,A -85,B 0,C 180,E1 -6383.044,E2 -6383.044} C_VEL
LIN {X 0,Y 488.794,Z 349.645,A -85,B 0,C 180,E1 -6384.429,E2 -6384.429} C_VEL
LIN {X 0,Y 489.199,Z 341.324,A -85,B 0,C 180,E1 -6385.673,E2 -6385.673} C_VEL
LIN {X 0,Y 489.698,Z 331.334,A -85,B 0,C 180,E1 -6386.914,E2 -6386.914} C_VEL
LIN {X 0,Y 490.178,Z 320.216,A -85,B 0,C 180,E1 -6388.047,E2 -6388.047} C_VEL
LIN {X 0,Y 490.75,Z 307.782,A -85,B 0,C 180,E1 -6389.076,E2 -6389.076} C_VEL
LIN {X 0,Y 491.351,Z 295.433,A -85,B 0,C 180,E1 -6389.896,E2 -6389.896} C_VEL
LIN {X 0,Y 491.819,Z 282.822,A -85,B 0,C 180,E1 -6390.562,E2 -6390.562} C_VEL
LIN {X 0,Y 492.156,Z 268.866,A -85,B 0,C 180,E1 -6391.12,E2 -6391.12} C_VEL
LIN {X 0,Y 492.463,Z 254.085,A -85,B 0,C 180,E1 -6391.522,E2 -6391.522} C_VEL
LIN {X 0,Y 493.298,Z 161.301,A -85,B 0,C 180,E1 -6392.917,E2 -6392.917} C_VEL
LIN {X 0,Y 493.409,Z 131.51,A -85,B 0,C 180,E1 -6393.363,E2 -6393.363} C_VEL
LIN {X 0,Y 490.298,Z 116.873,A -85,B 0,C 180,E1 -6393.71,E2 -6393.71} C_VEL
LIN {X 0,Y 490.79,Z 105.42,A -85,B 0,C 180,E1 -6395.752,E2 -6395.752} C_VEL
LIN {X 0,Y 488.837,Z 95.222,A -85,B 0,C 180,E1 -6397.714,E2 -6397.714} C_VEL
LIN {X 0,Y 488.725,Z 95.232,A -85,B 0,C 180,E1 -6400.773,E2 -6400.773} C_VEL
LIN {X 0,Y 488.754,Z 95.233,A -85,B 0,C 180,E1 -6403.3,E2 -6403.3} C_VEL
LIN {X 0,Y 488.737,Z 95.232,A -85,B 0,C 180,E1 -6405.855,E2 -6405.855} C_VEL
LIN {X 0,Y 488.729,Z 95.227,A -85,B 0,C 180,E1 -6408.442,E2 -6408.442} C_VEL
LIN {X 0,Y 488.706,Z 95.233,A -85,B 0,C 180,E1 -6411.069,E2 -6411.069} C_VEL
LIN {X 0,Y 488.682,Z 95.237,A -85,B 0,C 180,E1 -6413.745,E2 -6413.745} C_VEL
LIN {X 0,Y 488.762,Z 95.227,A -85,B 0,C 180,E1 -6416.946,E2 -6416.946} C_VEL
LIN {X 0,Y 488.689,Z 95.232,A -85,B 0,C 180,E1 -6420.367,E2 -6420.367} C_VEL
LIN {X 0,Y 488.704,Z 95.234,A -85,B 0,C 180,E1 -6423.487,E2 -6423.487} C_VEL
LIN {X 0,Y 488.673,Z 95.235,A -85,B 0,C 180,E1 -6426.36,E2 -6426.36} C_VEL
LIN {X 0,Y 488.726,Z 95.231,A -85,B 0,C 180,E1 -6429.25,E2 -6429.25} C_VEL
LIN {X 0,Y 488.707,Z 95.234,A -85,B 0,C 180,E1 -6432.522,E2 -6432.522} C_VEL
LIN {X 0,Y 488.696,Z 95.234,A -85,B 0,C 180,E1 -6435.203,E2 -6435.203} C_VEL
LIN {X 0,Y 488.714,Z 95.229,A -85,B 0,C 180,E1 -6437.482,E2 -6437.482} C_VEL
LIN {X 0,Y 488.726,Z 95.233,A -85,B 0,C 180,E1 -6440.753,E2 -6440.753} C_VEL
LIN {X 0,Y 488.662,Z 95.237,A -85,B 0,C 180,E1 -6443.871,E2 -6443.871} C_VEL
LIN {X 0,Y 488.713,Z 95.231,A -85,B 0,C 180,E1 -6446.88,E2 -6446.88} C_VEL
LIN {X 0,Y 488.709,Z 95.232,A -85,B 0,C 180,E1 -6449.784,E2 -6449.784} C_VEL
LIN {X 0,Y 488.775,Z 95.222,A -85,B 0,C 180,E1 -6453.057,E2 -6453.057} C_VEL
LIN {X 0,Y 488.695,Z 95.237,A -85,B 0,C 180,E1 -6456.259,E2 -6456.259} C_VEL
LIN {X 0,Y 488.727,Z 95.228,A -85,B 0,C 180,E1 -6459.178,E2 -6459.178} C_VEL
LIN {X 0,Y 488.739,Z 95.23,A -85,B 0,C 180,E1 -6461.63,E2 -6461.63} C_VEL
LIN {X 0,Y 488.744,Z 95.225,A -85,B 0,C 180,E1 -6465.002,E2 -6465.002} C_VEL
LIN {X 0,Y 488.815,Z 95.217,A -85,B 0,C 180,E1 -6468.391,E2 -6468.391} C_VEL
LIN {X 0,Y 488.805,Z 95.224,A -85,B 0,C 180,E1 -6471.736,E2 -6471.736} C_VEL
LIN {X 0,Y 488.85,Z 95.213,A -85,B 0,C 180,E1 -6474.227,E2 -6474.227} C_VEL
LIN {X 0,Y 488.951,Z 95.206,A -85,B 0,C 180,E1 -6477.531,E2 -6477.531} C_VEL
LIN {X 0,Y 488.958,Z 95.2,A -85,B 0,C 180,E1 -6480.003,E2 -6480.003} C_VEL
LIN {X 0,Y 488.952,Z 95.2,A -85,B 0,C 180,E1 -6482.474,E2 -6482.474} C_VEL
LIN {X 0,Y 488.847,Z 95.214,A -85,B 0,C 180,E1 -6485.778,E2 -6485.778} C_VEL
LIN {X 0,Y 488.81,Z 95.217,A -85,B 0,C 180,E1 -6488.269,E2 -6488.269} C_VEL
LIN {X 0,Y 488.798,Z 95.22,A -85,B 0,C 180,E1 -6491.615,E2 -6491.615} C_VEL
LIN {X 0,Y 488.755,Z 95.231,A -85,B 0,C 180,E1 -6495.003,E2 -6495.003} C_VEL
LIN {X 0,Y 488.749,Z 95.228,A -85,B 0,C 180,E1 -6498.445,E2 -6498.445} C_VEL
LIN {X 0,Y 488.703,Z 95.234,A -85,B 0,C 180,E1 -6501.073,E2 -6501.073} C_VEL
LIN {X 0,Y 488.689,Z 95.232,A -85,B 0,C 180,E1 -6503.748,E2 -6503.748} C_VEL
LIN {X 0,Y 488.796,Z 95.222,A -85,B 0,C 180,E1 -6506.948,E2 -6506.948} C_VEL
LIN {X 0,Y 488.707,Z 95.238,A -85,B 0,C 180,E1 -6510.365,E2 -6510.365} C_VEL
LIN {X 0,Y 488.733,Z 95.227,A -85,B 0,C 180,E1 -6513.486,E2 -6513.486} C_VEL
LIN {X 0,Y 488.685,Z 95.239,A -85,B 0,C 180,E1 -6516.357,E2 -6516.357} C_VEL
LIN {X 0,Y 488.699,Z 95.231,A -85,B 0,C 180,E1 -6519.256,E2 -6519.256} C_VEL
LIN {X 0,Y 488.706,Z 95.233,A -85,B 0,C 180,E1 -6521.602,E2 -6521.602} C_VEL
LIN {X 0,Y 488.711,Z 95.23,A -85,B 0,C 180,E1 -6524.803,E2 -6524.803} C_VEL
LIN {X 0,Y 488.691,Z 95.235,A -85,B 0,C 180,E1 -6527.476,E2 -6527.476} C_VEL
LIN {X 0,Y 488.733,Z 95.233,A -85,B 0,C 180,E1 -6529.678,E2 -6529.678} C_VEL
LIN {X 0,Y 488.679,Z 95.234,A -85,B 0,C 180,E1 -6532.843,E2 -6532.843} C_VEL
LIN {X 0,Y 488.73,Z 95.234,A -85,B 0,C 180,E1 -6535.889,E2 -6535.889} C_VEL
LIN {X 0,Y 488.691,Z 95.235,A -85,B 0,C 180,E1 -6538.822,E2 -6538.822} C_VEL
LIN {X 0,Y 488.745,Z 95.234,A -85,B 0,C 180,E1 -6541.673,E2 -6541.673} C_VEL
LIN {X 0,Y 488.78,Z 95.311,A -85,B 0,C 180,E1 -6543.01,E2 -6543.01} C_VEL
LIN {X 0,Y 491.283,Z 107.259,A -85,B 0,C 180,E1 -6545.04,E2 -6545.04} C_VEL
LIN {X 0,Y 491.386,Z 111.705,A -85,B 0,C 180,E1 -6545.744,E2 -6545.744} C_VEL
LIN {X 0,Y 490.516,Z 132.971,A -85,B 0,C 180,E1 -6549.012,E2 -6549.012} C_VEL
LIN {X 0,Y 490.231,Z 141.631,A -85,B 0,C 180,E1 -6550.317,E2 -6550.317} C_VEL
LIN {X 0,Y 493.361,Z 159.626,A -85,B 0,C 180,E1 -6550.711,E2 -6550.711} C_VEL
LIN {X 0,Y 492.385,Z 279.643,A -85,B 0,C 180,E1 -6552.506,E2 -6552.506} C_VEL
LIN {X 0,Y 492.009,Z 294.412,A -85,B 0,C 180,E1 -6552.899,E2 -6552.899} C_VEL
LIN {X 0,Y 491.606,Z 308.665,A -85,B 0,C 180,E1 -6553.461,E2 -6553.461} C_VEL
LIN {X 0,Y 491.066,Z 321.3,A -85,B 0,C 180,E1 -6554.119,E2 -6554.119} C_VEL
LIN {X 0,Y 490.526,Z 333.873,A -85,B 0,C 180,E1 -6554.95,E2 -6554.95} C_VEL
LIN {X 0,Y 489.924,Z 345.386,A -85,B 0,C 180,E1 -6555.886,E2 -6555.886} C_VEL
LIN {X 0,Y 489.457,Z 355.943,A -85,B 0,C 180,E1 -6556.931,E2 -6556.931} C_VEL
LIN {X 0,Y 489.072,Z 365.55,A -85,B 0,C 180,E1 -6558.071,E2 -6558.071} C_VEL
LIN {X 0,Y 488.655,Z 375.095,A -85,B 0,C 180,E1 -6559.435,E2 -6559.435} C_VEL
LIN {X 0,Y 488.322,Z 383.388,A -85,B 0,C 180,E1 -6560.892,E2 -6560.892} C_VEL
LIN {X 0,Y 488.144,Z 389.183,A -85,B 0,C 180,E1 -6562.14,E2 -6562.14} C_VEL
LIN {X 0,Y 488.023,Z 394.516,A -85,B 0,C 180,E1 -6563.553,E2 -6563.553} C_VEL
LIN {X 0,Y 487.958,Z 398.858,A -85,B 0,C 180,E1 -6565.044,E2 -6565.044} C_VEL
LIN {X 0,Y 487.956,Z 402.28,A -85,B 0,C 180,E1 -6566.698,E2 -6566.698} C_VEL
LIN {X 0,Y 487.89,Z 404.301,A -85,B 0,C 180,E1 -6568.35,E2 -6568.35} C_VEL
LIN {X 0,Y 487.822,Z 404.968,A -85,B 0,C 180,E1 -6570.001,E2 -6570.001} C_VEL
LIN {X 0,Y 487.89,Z 404.297,A -85,B 0,C 180,E1 -6571.652,E2 -6571.652} C_VEL
LIN {X 0,Y 487.957,Z 402.273,A -85,B 0,C 180,E1 -6573.304,E2 -6573.304} C_VEL
LIN {X 0,Y 487.959,Z 398.847,A -85,B 0,C 180,E1 -6574.959,E2 -6574.959} C_VEL
LIN {X 0,Y 488.04,Z 393.921,A -85,B 0,C 180,E1 -6576.617,E2 -6576.617} C_VEL
LIN {X 0,Y 488.218,Z 387.351,A -85,B 0,C 180,E1 -6578.278,E2 -6578.278} C_VEL
LIN {X 0,Y 488.449,Z 380.043,A -85,B 0,C 180,E1 -6579.735,E2 -6579.735} C_VEL
LIN {X 0,Y 488.853,Z 370.997,A -85,B 0,C 180,E1 -6581.192,E2 -6581.192} C_VEL
LIN {X 0,Y 489.241,Z 361.516,A -85,B 0,C 180,E1 -6582.445,E2 -6582.445} C_VEL
LIN {X 0,Y 489.733,Z 351.041,A -85,B 0,C 180,E1 -6583.592,E2 -6583.592} C_VEL
LIN {X 0,Y 490.256,Z 339.496,A -85,B 0,C 180,E1 -6584.636,E2 -6584.636} C_VEL
LIN {X 0,Y 490.888,Z 326.704,A -85,B 0,C 180,E1 -6585.573,E2 -6585.573} C_VEL
LIN {X 0,Y 491.435,Z 314.52,A -85,B 0,C 180,E1 -6586.285,E2 -6586.285} C_VEL
LIN {X 0,Y 491.881,Z 301.17,A -85,B 0,C 180,E1 -6586.894,E2 -6586.894} C_VEL
LIN {X 0,Y 492.312,Z 287.089,A -85,B 0,C 180,E1 -6587.357,E2 -6587.357} C_VEL
LIN {X 0,Y 492.613,Z 273.223,A -85,B 0,C 180,E1 -6587.649,E2 -6587.649} C_VEL
LIN {X 0,Y 493.525,Z 159.632,A -85,B 0,C 180,E1 -6589.341,E2 -6589.341} C_VEL
LIN {X 0,Y 490.274,Z 141.165,A -85,B 0,C 180,E1 -6589.79,E2 -6589.79} C_VEL
LIN {X 0,Y 491.169,Z 119.356,A -85,B 0,C 180,E1 -6593.173,E2 -6593.173} C_VEL
LIN {X 0,Y 491.657,Z 109.535,A -85,B 0,C 180,E1 -6594.717,E2 -6594.717} C_VEL
LIN {X 0,Y 490.053,Z 101.153,A -85,B 0,C 180,E1 -6596.168,E2 -6596.168} C_VEL
LIN {X 0,Y 488.779,Z 95.226,A -85,B 0,C 180,E1 -6597.262,E2 -6597.262} C_VEL
LIN {X 0,Y 488.719,Z 95.235,A -85,B 0,C 180,E1 -6600.363,E2 -6600.363} C_VEL
LIN {X 0,Y 488.741,Z 95.232,A -85,B 0,C 180,E1 -6603.483,E2 -6603.483} C_VEL
LIN {X 0,Y 488.685,Z 95.24,A -85,B 0,C 180,E1 -6606.353,E2 -6606.353} C_VEL
LIN {X 0,Y 488.709,Z 95.232,A -85,B 0,C 180,E1 -6609.255,E2 -6609.255} C_VEL
LIN {X 0,Y 488.71,Z 95.232,A -85,B 0,C 180,E1 -6611.598,E2 -6611.598} C_VEL
LIN {X 0,Y 488.714,Z 95.23,A -85,B 0,C 180,E1 -6614.803,E2 -6614.803} C_VEL
LIN {X 0,Y 488.705,Z 95.236,A -85,B 0,C 180,E1 -6617.474,E2 -6617.474} C_VEL
LIN {X 0,Y 488.716,Z 95.228,A -85,B 0,C 180,E1 -6619.673,E2 -6619.673} C_VEL
LIN {X 0,Y 488.682,Z 95.233,A -85,B 0,C 180,E1 -6622.84,E2 -6622.84} C_VEL
LIN {X 0,Y 488.736,Z 95.229,A -85,B 0,C 180,E1 -6625.886,E2 -6625.886} C_VEL
LIN {X 0,Y 488.703,Z 95.232,A -85,B 0,C 180,E1 -6628.819,E2 -6628.819} C_VEL
LIN {X 0,Y 488.725,Z 95.229,A -85,B 0,C 180,E1 -6631.668,E2 -6631.668} C_VEL
LIN {X 0,Y 488.726,Z 95.23,A -85,B 0,C 180,E1 -6634.441,E2 -6634.441} C_VEL
LIN {X 0,Y 488.734,Z 95.234,A -85,B 0,C 180,E1 -6637.152,E2 -6637.152} C_VEL
LIN {X 0,Y 488.735,Z 95.223,A -85,B 0,C 180,E1 -6639.809,E2 -6639.809} C_VEL
LIN {X 0,Y 488.722,Z 95.232,A -85,B 0,C 180,E1 -6642.421,E2 -6642.421} C_VEL
LIN {X 0,Y 488.769,Z 95.228,A -85,B 0,C 180,E1 -6644.998,E2 -6644.998} C_VEL
LIN {X 0,Y 488.816,Z 95.219,A -85,B 0,C 180,E1 -6648.385,E2 -6648.385} C_VEL
LIN {X 0,Y 488.79,Z 95.22,A -85,B 0,C 180,E1 -6651.731,E2 -6651.731} C_VEL
LIN {X 0,Y 488.837,Z 95.219,A -85,B 0,C 180,E1 -6654.222,E2 -6654.222} C_VEL
LIN {X 0,Y 488.961,Z 95.196,A -85,B 0,C 180,E1 -6657.526,E2 -6657.526} C_VEL
LIN {X 0,Y 488.976,Z 95.204,A -85,B 0,C 180,E1 -6659.997,E2 -6659.997} C_VEL
LIN {X 0,Y 488.959,Z 95.202,A -85,B 0,C 180,E1 -6662.469,E2 -6662.469} C_VEL
LIN {X 0,Y 488.842,Z 95.216,A -85,B 0,C 180,E1 -6665.773,E2 -6665.773} C_VEL
LIN {X 0,Y 488.788,Z 95.222,A -85,B 0,C 180,E1 -6668.264,E2 -6668.264} C_VEL
LIN {X 0,Y 488.807,Z 95.225,A -85,B 0,C 180,E1 -6671.609,E2 -6671.609} C_VEL
LIN {X 0,Y 488.76,Z 95.226,A -85,B 0,C 180,E1 -6674.997,E2 -6674.997} C_VEL
LIN {X 0,Y 488.743,Z 95.227,A -85,B 0,C 180,E1 -6678.439,E2 -6678.439} C_VEL
LIN {X 0,Y 488.703,Z 95.234,A -85,B 0,C 180,E1 -6681.067,E2 -6681.067} C_VEL
LIN {X 0,Y 488.666,Z 95.238,A -85,B 0,C 180,E1 -6683.743,E2 -6683.743} C_VEL
LIN {X 0,Y 488.74,Z 95.23,A -85,B 0,C 180,E1 -6686.93,E2 -6686.93} C_VEL
LIN {X 0,Y 488.713,Z 95.226,A -85,B 0,C 180,E1 -6689.267,E2 -6689.267} C_VEL
LIN {X 0,Y 488.691,Z 95.234,A -85,B 0,C 180,E1 -6692.143,E2 -6692.143} C_VEL
LIN {X 0,Y 488.701,Z 95.237,A -85,B 0,C 180,E1 -6695.112,E2 -6695.112} C_VEL
LIN {X 0,Y 488.661,Z 95.235,A -85,B 0,C 180,E1 -6698.197,E2 -6698.197} C_VEL
LIN {X 0,Y 488.702,Z 95.237,A -85,B 0,C 180,E1 -6700.341,E2 -6700.341} C_VEL
LIN {X 0,Y 488.665,Z 95.239,A -85,B 0,C 180,E1 -6703.651,E2 -6703.651} C_VEL
LIN {X 0,Y 488.657,Z 95.246,A -85,B 0,C 180,E1 -6706.341,E2 -6706.341} C_VEL
LIN {X 0,Y 488.68,Z 95.246,A -85,B 0,C 180,E1 -6709.67,E2 -6709.67} C_VEL
LIN {X 0,Y 488.714,Z 95.38,A -85,B 0,C 180,E1 -6710.178,E2 -6710.178} C_VEL
LIN {X 0,Y 490.775,Z 105.866,A -85,B 0,C 180,E1 -6712.259,E2 -6712.259} C_VEL
LIN {X 0,Y 490.566,Z 114.313,A -85,B 0,C 180,E1 -6713.801,E2 -6713.801} C_VEL
LIN {X 0,Y 490.492,Z 117.105,A -85,B 0,C 180,E1 -6714.301,E2 -6714.301} C_VEL
LIN {X 0,Y 493.719,Z 132.861,A -85,B 0,C 180,E1 -6714.688,E2 -6714.688} C_VEL
LIN {X 0,Y 493.167,Z 192.127,A -85,B 0,C 180,E1 -6715.57,E2 -6715.57} C_VEL
LIN {X 0,Y 492.38,Z 197.979,A -85,B 0,C 180,E1 -6715.627,E2 -6715.627} C_VEL
LIN {X 0,Y 486.836,Z 217.022,A -85,B 0,C 180,E1 -6715.687,E2 -6715.687} C_VEL
LIN {X 0,Y 486.261,Z 222.863,A -85,B 0,C 180,E1 -6715.753,E2 -6715.753} C_VEL
LIN {X 0,Y 485.93,Z 254.483,A -85,B 0,C 180,E1 -6716.256,E2 -6716.256} C_VEL
LIN {X 0,Y 485.592,Z 268.889,A -85,B 0,C 180,E1 -6716.654,E2 -6716.654} C_VEL
LIN {X 0,Y 485.193,Z 281.861,A -85,B 0,C 180,E1 -6717.172,E2 -6717.172} C_VEL
LIN {X 0,Y 484.608,Z 295.846,A -85,B 0,C 180,E1 -6717.916,E2 -6717.916} C_VEL
LIN {X 0,Y 484.046,Z 308.564,A -85,B 0,C 180,E1 -6718.785,E2 -6718.785} C_VEL
LIN {X 0,Y 483.436,Z 320.29,A -85,B 0,C 180,E1 -6719.776,E2 -6719.776} C_VEL
LIN {X 0,Y 482.851,Z 330.625,A -85,B 0,C 180,E1 -6720.837,E2 -6720.837} C_VEL
LIN {X 0,Y 482.356,Z 339.846,A -85,B 0,C 180,E1 -6721.972,E2 -6721.972} C_VEL
LIN {X 0,Y 481.876,Z 349.176,A -85,B 0,C 180,E1 -6723.353,E2 -6723.353} C_VEL
LIN {X 0,Y 481.505,Z 357.15,A -85,B 0,C 180,E1 -6724.805,E2 -6724.805} C_VEL
LIN {X 0,Y 481.2,Z 363.833,A -85,B 0,C 180,E1 -6726.318,E2 -6726.318} C_VEL
LIN {X 0,Y 481.077,Z 368.641,A -85,B 0,C 180,E1 -6727.676,E2 -6727.676} C_VEL
LIN {X 0,Y 480.944,Z 372.912,A -85,B 0,C 180,E1 -6729.252,E2 -6729.252} C_VEL
LIN {X 0,Y 480.794,Z 375.104,A -85,B 0,C 180,E1 -6730.353,E2 -6730.353} C_VEL
LIN {X 0,Y 480.761,Z 377.426,A -85,B 0,C 180,E1 -6732.121,E2 -6732.121} C_VEL
LIN {X 0,Y 480.681,Z 378.283,A -85,B 0,C 180,E1 -6733.87,E2 -6733.87} C_VEL
LIN {X 0,Y 480.746,Z 377.717,A -85,B 0,C 180,E1 -6735.609,E2 -6735.609} C_VEL
LIN {X 0,Y 480.789,Z 375.732,A -85,B 0,C 180,E1 -6737.333,E2 -6737.333} C_VEL
LIN {X 0,Y 480.904,Z 372.305,A -85,B 0,C 180,E1 -6739.047,E2 -6739.047} C_VEL
LIN {X 0,Y 481.055,Z 367.38,A -85,B 0,C 180,E1 -6740.751,E2 -6740.751} C_VEL
LIN {X 0,Y 481.235,Z 362.632,A -85,B 0,C 180,E1 -6742.024,E2 -6742.024} C_VEL
LIN {X 0,Y 481.534,Z 355.766,A -85,B 0,C 180,E1 -6743.504,E2 -6743.504} C_VEL
LIN {X 0,Y 481.896,Z 347.289,A -85,B 0,C 180,E1 -6744.979,E2 -6744.979} C_VEL
LIN {X 0,Y 482.354,Z 338.455,A -85,B 0,C 180,E1 -6746.239,E2 -6746.239} C_VEL
LIN {X 0,Y 482.902,Z 327.797,A -85,B 0,C 180,E1 -6747.496,E2 -6747.496} C_VEL
LIN {X 0,Y 483.518,Z 315.873,A -85,B 0,C 180,E1 -6748.645,E2 -6748.645} C_VEL
LIN {X 0,Y 484.096,Z 303.842,A -85,B 0,C 180,E1 -6749.583,E2 -6749.583} C_VEL
LIN {X 0,Y 484.692,Z 290.384,A -85,B 0,C 180,E1 -6750.415,E2 -6750.415} C_VEL
LIN {X 0,Y 485.169,Z 277.153,A -85,B 0,C 180,E1 -6751.046,E2 -6751.046} C_VEL
LIN {X 0,Y 485.534,Z 263.081,A -85,B 0,C 180,E1 -6751.537,E2 -6751.537} C_VEL
LIN {X 0,Y 485.723,Z 248.713,A -85,B 0,C 180,E1 -6751.864,E2 -6751.864} C_VEL
LIN {X 0,Y 486.814,Z 133.105,A -85,B 0,C 180,E1 -6753.598,E2 -6753.598} C_VEL
LIN {X 0,Y 483.418,Z 116.956,A -85,B 0,C 180,E1 -6754.003,E2 -6754.003} C_VEL
LIN {X 0,Y 483.839,Z 106.811,A -85,B 0,C 180,E1 -6755.835,E2 -6755.835} C_VEL
LIN {X 0,Y 481.806,Z 96.097,A -85,B 0,C 180,E1 -6757.922,E2 -6757.922} C_VEL
LIN {X 0,Y 481.759,Z 96.104,A -85,B 0,C 180,E1 -6761.783,E2 -6761.783} C_VEL
LIN {X 0,Y 481.739,Z 96.101,A -85,B 0,C 180,E1 -6765.223,E2 -6765.223} C_VEL
LIN {X 0,Y 481.68,Z 96.106,A -85,B 0,C 180,E1 -6768.722,E2 -6768.722} C_VEL
LIN {X 0,Y 481.643,Z 96.117,A -85,B 0,C 180,E1 -6771.393,E2 -6771.393} C_VEL
LIN {X 0,Y 481.663,Z 96.108,A -85,B 0,C 180,E1 -6774.112,E2 -6774.112} C_VEL
LIN {X 0,Y 481.715,Z 96.107,A -85,B 0,C 180,E1 -6777.142,E2 -6777.142} C_VEL
LIN {X 0,Y 481.655,Z 96.11,A -85,B 0,C 180,E1 -6779.741,E2 -6779.741} C_VEL
LIN {X 0,Y 481.641,Z 96.113,A -85,B 0,C 180,E1 -6782.675,E2 -6782.675} C_VEL
LIN {X 0,Y 481.624,Z 96.113,A -85,B 0,C 180,E1 -6785.709,E2 -6785.709} C_VEL
LIN {X 0,Y 481.684,Z 96.112,A -85,B 0,C 180,E1 -6788.856,E2 -6788.856} C_VEL
LIN {X 0,Y 481.646,Z 96.11,A -85,B 0,C 180,E1 -6792.159,E2 -6792.159} C_VEL
LIN {X 0,Y 481.662,Z 96.112,A -85,B 0,C 180,E1 -6794.455,E2 -6794.455} C_VEL
LIN {X 0,Y 481.705,Z 96.108,A -85,B 0,C 180,E1 -6796.842,E2 -6796.842} C_VEL
LIN {X 0,Y 481.684,Z 96.107,A -85,B 0,C 180,E1 -6800.066,E2 -6800.066} C_VEL
LIN {X 0,Y 481.608,Z 96.114,A -85,B 0,C 180,E1 -6803.377,E2 -6803.377} C_VEL
LIN {X 0,Y 481.682,Z 96.113,A -85,B 0,C 180,E1 -6806.332,E2 -6806.332} C_VEL
LIN {X 0,Y 481.634,Z 96.111,A -85,B 0,C 180,E1 -6809.418,E2 -6809.418} C_VEL
LIN {X 0,Y 481.679,Z 96.113,A -85,B 0,C 180,E1 -6812.171,E2 -6812.171} C_VEL
LIN {X 0,Y 481.702,Z 96.103,A -85,B 0,C 180,E1 -6814.973,E2 -6814.973} C_VEL
LIN {X 0,Y 481.655,Z 96.112,A -85,B 0,C 180,E1 -6817.709,E2 -6817.709} C_VEL
LIN {X 0,Y 481.689,Z 96.107,A -85,B 0,C 180,E1 -6820.396,E2 -6820.396} C_VEL
LIN {X 0,Y 481.674,Z 96.106,A -85,B 0,C 180,E1 -6823.037,E2 -6823.037} C_VEL
LIN {X 0,Y 481.674,Z 96.112,A -85,B 0,C 180,E1 -6825.642,E2 -6825.642} C_VEL
LIN {X 0,Y 481.779,Z 96.095,A -85,B 0,C 180,E1 -6828.219,E2 -6828.219} C_VEL
LIN {X 0,Y 481.751,Z 96.105,A -85,B 0,C 180,E1 -6831.615,E2 -6831.615} C_VEL
LIN {X 0,Y 481.81,Z 96.09,A -85,B 0,C 180,E1 -6834.142,E2 -6834.142} C_VEL
LIN {X 0,Y 481.918,Z 96.083,A -85,B 0,C 180,E1 -6837.495,E2 -6837.495} C_VEL
LIN {X 0,Y 481.929,Z 96.075,A -85,B 0,C 180,E1 -6840.003,E2 -6840.003} C_VEL
LIN {X 0,Y 481.919,Z 96.076,A -85,B 0,C 180,E1 -6842.51,E2 -6842.51} C_VEL
LIN {X 0,Y 481.808,Z 96.09,A -85,B 0,C 180,E1 -6845.863,E2 -6845.863} C_VEL
LIN {X 0,Y 481.755,Z 96.097,A -85,B 0,C 180,E1 -6848.391,E2 -6848.391} C_VEL
LIN {X 0,Y 481.743,Z 96.098,A -85,B 0,C 180,E1 -6851.787,E2 -6851.787} C_VEL
LIN {X 0,Y 481.736,Z 96.102,A -85,B 0,C 180,E1 -6855.227,E2 -6855.227} C_VEL
LIN {X 0,Y 481.707,Z 96.11,A -85,B 0,C 180,E1 -6858.724,E2 -6858.724} C_VEL
LIN {X 0,Y 481.642,Z 96.111,A -85,B 0,C 180,E1 -6861.397,E2 -6861.397} C_VEL
LIN {X 0,Y 481.673,Z 96.108,A -85,B 0,C 180,E1 -6864.115,E2 -6864.115} C_VEL
LIN {X 0,Y 481.749,Z 96.098,A -85,B 0,C 180,E1 -6867.143,E2 -6867.143} C_VEL
LIN {X 0,Y 481.676,Z 96.107,A -85,B 0,C 180,E1 -6869.743,E2 -6869.743} C_VEL
LIN {X 0,Y 481.67,Z 96.11,A -85,B 0,C 180,E1 -6872.676,E2 -6872.676} C_VEL
LIN {X 0,Y 481.639,Z 96.112,A -85,B 0,C 180,E1 -6875.711,E2 -6875.711} C_VEL
LIN {X 0,Y 481.668,Z 96.107,A -85,B 0,C 180,E1 -6878.861,E2 -6878.861} C_VEL
LIN {X 0,Y 481.652,Z 96.115,A -85,B 0,C 180,E1 -6881.915,E2 -6881.915} C_VEL
LIN {X 0,Y 481.659,Z 96.11,A -85,B 0,C 180,E1 -6884.459,E2 -6884.459} C_VEL
LIN {X 0,Y 481.647,Z 96.118,A -85,B 0,C 180,E1 -6887.841,E2 -6887.841} C_VEL
LIN {X 0,Y 481.661,Z 96.108,A -85,B 0,C 180,E1 -6890.656,E2 -6890.656} C_VEL
LIN {X 0,Y 481.627,Z 96.116,A -85,B 0,C 180,E1 -6893.378,E2 -6893.378} C_VEL
LIN {X 0,Y 481.695,Z 96.104,A -85,B 0,C 180,E1 -6896.331,E2 -6896.331} C_VEL
LIN {X 0,Y 481.65,Z 96.116,A -85,B 0,C 180,E1 -6899.42,E2 -6899.42} C_VEL
LIN {X 0,Y 481.71,Z 96.108,A -85,B 0,C 180,E1 -6902.56,E2 -6902.56} C_VEL
LIN {X 0,Y 481.759,Z 96.286,A -85,B 0,C 180,E1 -6902.803,E2 -6902.803} C_VEL
LIN {X 0,Y 484.525,Z 109.817,A -85,B 0,C 180,E1 -6905.126,E2 -6905.126} C_VEL
LIN {X 0,Y 483.855,Z 126.949,A -85,B 0,C 180,E1 -6907.813,E2 -6907.813} C_VEL
LIN {X 0,Y 483.273,Z 141.28,A -85,B 0,C 180,E1 -6910.029,E2 -6910.029} C_VEL
LIN {X 0,Y 486.658,Z 161.547,A -85,B 0,C 180,E1 -6910.482,E2 -6910.482} C_VEL
LIN {X 0,Y 485.591,Z 278.798,A -85,B 0,C 180,E1 -6912.253,E2 -6912.253} C_VEL
LIN {X 0,Y 485.255,Z 292.978,A -85,B 0,C 180,E1 -6912.624,E2 -6912.624} C_VEL
LIN {X 0,Y 484.803,Z 306.618,A -85,B 0,C 180,E1 -6913.147,E2 -6913.147} C_VEL
LIN {X 0,Y 484.286,Z 319.354,A -85,B 0,C 180,E1 -6913.798,E2 -6913.798} C_VEL
LIN {X 0,Y 483.687,Z 332.056,A -85,B 0,C 180,E1 -6914.624,E2 -6914.624} C_VEL
LIN {X 0,Y 483.079,Z 343.857,A -85,B 0,C 180,E1 -6915.575,E2 -6915.575} C_VEL
LIN {X 0,Y 482.492,Z 355.637,A -85,B 0,C 180,E1 -6916.739,E2 -6916.739} C_VEL
LIN {X 0,Y 482.067,Z 365.611,A -85,B 0,C 180,E1 -6917.938,E2 -6917.938} C_VEL
LIN {X 0,Y 481.626,Z 374.848,A -85,B 0,C 180,E1 -6919.279,E2 -6919.279} C_VEL
LIN {X 0,Y 481.281,Z 383.165,A -85,B 0,C 180,E1 -6920.758,E2 -6920.758} C_VEL
LIN {X 0,Y 481.074,Z 388.966,A -85,B 0,C 180,E1 -6922.024,E2 -6922.024} C_VEL
LIN {X 0,Y 480.913,Z 394.768,A -85,B 0,C 180,E1 -6923.594,E2 -6923.594} C_VEL
LIN {X 0,Y 480.886,Z 398.652,A -85,B 0,C 180,E1 -6924.971,E2 -6924.971} C_VEL
LIN {X 0,Y 480.862,Z 402.077,A -85,B 0,C 180,E1 -6926.65,E2 -6926.65} C_VEL
LIN {X 0,Y 480.791,Z 404.102,A -85,B 0,C 180,E1 -6928.326,E2 -6928.326} C_VEL
LIN {X 0,Y 480.745,Z 404.773,A -85,B 0,C 180,E1 -6930.001,E2 -6930.001} C_VEL
LIN {X 0,Y 480.792,Z 404.104,A -85,B 0,C 180,E1 -6931.676,E2 -6931.676} C_VEL
LIN {X 0,Y 480.863,Z 402.083,A -85,B 0,C 180,E1 -6933.353,E2 -6933.353} C_VEL
LIN {X 0,Y 480.888,Z 398.659,A -85,B 0,C 180,E1 -6935.032,E2 -6935.032} C_VEL
LIN {X 0,Y 480.963,Z 393.734,A -85,B 0,C 180,E1 -6936.714,E2 -6936.714} C_VEL
LIN {X 0,Y 481.135,Z 387.175,A -85,B 0,C 180,E1 -6938.4,E2 -6938.4} C_VEL
LIN {X 0,Y 481.404,Z 379.883,A -85,B 0,C 180,E1 -6939.878,E2 -6939.878} C_VEL
LIN {X 0,Y 481.846,Z 370.866,A -85,B 0,C 180,E1 -6941.357,E2 -6941.357} C_VEL
LIN {X 0,Y 482.26,Z 361.41,A -85,B 0,C 180,E1 -6942.628,E2 -6942.628} C_VEL
LIN {X 0,Y 482.794,Z 350.954,A -85,B 0,C 180,E1 -6943.791,E2 -6943.791} C_VEL
LIN {X 0,Y 483.367,Z 339.432,A -85,B 0,C 180,E1 -6944.849,E2 -6944.849} C_VEL
LIN {X 0,Y 484.021,Z 326.67,A -85,B 0,C 180,E1 -6945.799,E2 -6945.799} C_VEL
LIN {X 0,Y 484.671,Z 313.181,A -85,B 0,C 180,E1 -6946.592,E2 -6946.592} C_VEL
LIN {X 0,Y 485.127,Z 300.076,A -85,B 0,C 180,E1 -6947.185,E2 -6947.185} C_VEL
LIN {X 0,Y 485.579,Z 286.298,A -85,B 0,C 180,E1 -6947.636,E2 -6947.636} C_VEL
LIN {X 0,Y 485.919,Z 272.225,A -85,B 0,C 180,E1 -6947.928,E2 -6947.928} C_VEL
LIN {X 0,Y 486.894,Z 160.623,A -85,B 0,C 180,E1 -6949.615,E2 -6949.615} C_VEL
LIN {X 0,Y 483.346,Z 141.095,A -85,B 0,C 180,E1 -6950.087,E2 -6950.087} C_VEL
LIN {X 0,Y 484.294,Z 120.748,A -85,B 0,C 180,E1 -6953.289,E2 -6953.289} C_VEL
LIN {X 0,Y 484.797,Z 110.937,A -85,B 0,C 180,E1 -6954.861,E2 -6954.861} C_VEL
LIN {X 0,Y 482.097,Z 97.731,A -85,B 0,C 180,E1 -6957.218,E2 -6957.218} C_VEL
LIN {X 0,Y 481.719,Z 96.104,A -85,B 0,C 180,E1 -6957.547,E2 -6957.547} C_VEL
LIN {X 0,Y 481.655,Z 96.116,A -85,B 0,C 180,E1 -6960.711,E2 -6960.711} C_VEL
LIN {X 0,Y 481.687,Z 96.112,A -85,B 0,C 180,E1 -6963.729,E2 -6963.729} C_VEL
LIN {X 0,Y 481.632,Z 96.113,A -85,B 0,C 180,E1 -6966.748,E2 -6966.748} C_VEL
LIN {X 0,Y 481.67,Z 96.11,A -85,B 0,C 180,E1 -6969.942,E2 -6969.942} C_VEL
LIN {X 0,Y 481.639,Z 96.112,A -85,B 0,C 180,E1 -6973.146,E2 -6973.146} C_VEL
LIN {X 0,Y 481.667,Z 96.112,A -85,B 0,C 180,E1 -6975.641,E2 -6975.641} C_VEL
LIN {X 0,Y 481.662,Z 96.099,A -85,B 0,C 180,E1 -6978.957,E2 -6978.957} C_VEL
LIN {X 0,Y 481.662,Z 96.11,A -85,B 0,C 180,E1 -6981.993,E2 -6981.993} C_VEL
LIN {X 0,Y 481.697,Z 96.109,A -85,B 0,C 180,E1 -6985.317,E2 -6985.317} C_VEL
LIN {X 0,Y 481.657,Z 96.108,A -85,B 0,C 180,E1 -6988.31,E2 -6988.31} C_VEL
LIN {X 0,Y 481.687,Z 96.111,A -85,B 0,C 180,E1 -6991.216,E2 -6991.216} C_VEL
LIN {X 0,Y 481.681,Z 96.107,A -85,B 0,C 180,E1 -6994.04,E2 -6994.04} C_VEL
LIN {X 0,Y 481.688,Z 96.106,A -85,B 0,C 180,E1 -6996.811,E2 -6996.811} C_VEL
LIN {X 0,Y 481.707,Z 96.1,A -85,B 0,C 180,E1 -6999.501,E2 -6999.501} C_VEL
LIN {X 0,Y 481.701,Z 96.105,A -85,B 0,C 180,E1 -7002.156,E2 -7002.156} C_VEL
LIN {X 0,Y 481.752,Z 96.101,A -85,B 0,C 180,E1 -7004.774,E2 -7004.774} C_VEL
LIN {X 0,Y 481.762,Z 96.097,A -85,B 0,C 180,E1 -7008.213,E2 -7008.213} C_VEL
LIN {X 0,Y 481.746,Z 96.097,A -85,B 0,C 180,E1 -7011.609,E2 -7011.609} C_VEL
LIN {X 0,Y 481.796,Z 96.095,A -85,B 0,C 180,E1 -7014.137,E2 -7014.137} C_VEL
LIN {X 0,Y 481.927,Z 96.072,A -85,B 0,C 180,E1 -7017.49,E2 -7017.49} C_VEL
LIN {X 0,Y 481.947,Z 96.079,A -85,B 0,C 180,E1 -7019.997,E2 -7019.997} C_VEL
LIN {X 0,Y 481.926,Z 96.078,A -85,B 0,C 180,E1 -7022.505,E2 -7022.505} C_VEL
LIN {X 0,Y 481.801,Z 96.093,A -85,B 0,C 180,E1 -7025.858,E2 -7025.858} C_VEL
LIN {X 0,Y 481.743,Z 96.098,A -85,B 0,C 180,E1 -7028.386,E2 -7028.386} C_VEL
LIN {X 0,Y 481.753,Z 96.102,A -85,B 0,C 180,E1 -7031.782,E2 -7031.782} C_VEL
LIN {X 0,Y 481.741,Z 96.102,A -85,B 0,C 180,E1 -7035.221,E2 -7035.221} C_VEL
LIN {X 0,Y 481.705,Z 96.104,A -85,B 0,C 180,E1 -7038.718,E2 -7038.718} C_VEL
LIN {X 0,Y 481.642,Z 96.118,A -85,B 0,C 180,E1 -7041.391,E2 -7041.391} C_VEL
LIN {X 0,Y 481.644,Z 96.111,A -85,B 0,C 180,E1 -7044.111,E2 -7044.111} C_VEL
LIN {X 0,Y 481.707,Z 96.11,A -85,B 0,C 180,E1 -7047.128,E2 -7047.128} C_VEL
LIN {X 0,Y 481.668,Z 96.1,A -85,B 0,C 180,E1 -7049.737,E2 -7049.737} C_VEL
LIN {X 0,Y 481.659,Z 96.115,A -85,B 0,C 180,E1 -7052.671,E2 -7052.671} C_VEL
LIN {X 0,Y 481.622,Z 96.115,A -85,B 0,C 180,E1 -7055.706,E2 -7055.706} C_VEL
LIN {X 0,Y 481.651,Z 96.116,A -85,B 0,C 180,E1 -7058.856,E2 -7058.856} C_VEL
LIN {X 0,Y 481.635,Z 96.114,A -85,B 0,C 180,E1 -7061.909,E2 -7061.909} C_VEL
LIN {X 0,Y 481.636,Z 96.12,A -85,B 0,C 180,E1 -7064.454,E2 -7064.454} C_VEL
LIN {X 0,Y 481.621,Z 96.12,A -85,B 0,C 180,E1 -7067.835,E2 -7067.835} C_VEL
LIN {X 0,Y 481.656,Z 96.189,A -85,B 0,C 180,E1 -7069.894,E2 -7069.894} C_VEL
LIN {X 0,Y 483.835,Z 106.941,A -85,B 0,C 180,E1 -7072.068,E2 -7072.068} C_VEL
LIN {X 0,Y 483.799,Z 112.564,A -85,B 0,C 180,E1 -7073.12,E2 -7073.12} C_VEL
LIN {X 0,Y 483.629,Z 117.2,A -85,B 0,C 180,E1 -7073.973,E2 -7073.973} C_VEL
LIN {X 0,Y 487.089,Z 133.072,A -85,B 0,C 180,E1 -7074.394,E2 -7074.394} C_VEL
LIN {X 0,Y 486.261,Z 222.863,A -85,B 0,C 180,E1 -7075.753,E2 -7075.753} C_VEL
LIN {X 0,Y 485.671,Z 228.708,A -85,B 0,C 180,E1 -7075.816,E2 -7075.816} C_VEL
LIN {X 0,Y 480.022,Z 247.725,A -85,B 0,C 180,E1 -7075.876,E2 -7075.876} C_VEL
LIN {X 0,Y 479.253,Z 253.554,A -85,B 0,C 180,E1 -7075.954,E2 -7075.954} C_VEL
LIN {X 0,Y 478.906,Z 267.584,A -85,B 0,C 180,E1 -7076.329,E2 -7076.329} C_VEL
LIN {X 0,Y 478.523,Z 280.486,A -85,B 0,C 180,E1 -7076.832,E2 -7076.832} C_VEL
LIN {X 0,Y 477.939,Z 294.023,A -85,B 0,C 180,E1 -7077.538,E2 -7077.538} C_VEL
LIN {X 0,Y 477.295,Z 306.851,A -85,B 0,C 180,E1 -7078.397,E2 -7078.397} C_VEL
LIN {X 0,Y 476.629,Z 319.099,A -85,B 0,C 180,E1 -7079.421,E2 -7079.421} C_VEL
LIN {X 0,Y 475.959,Z 330.476,A -85,B 0,C 180,E1 -7080.588,E2 -7080.588} C_VEL
LIN {X 0,Y 475.432,Z 339.945,A -85,B 0,C 180,E1 -7081.767,E2 -7081.767} C_VEL
LIN {X 0,Y 474.882,Z 349.284,A -85,B 0,C 180,E1 -7083.166,E2 -7083.166} C_VEL
LIN {X 0,Y 474.506,Z 357.129,A -85,B 0,C 180,E1 -7084.609,E2 -7084.609} C_VEL
LIN {X 0,Y 474.183,Z 363.073,A -85,B 0,C 180,E1 -7085.946,E2 -7085.946} C_VEL
LIN {X 0,Y 474.039,Z 368.045,A -85,B 0,C 180,E1 -7087.326,E2 -7087.326} C_VEL
LIN {X 0,Y 473.913,Z 371.951,A -85,B 0,C 180,E1 -7088.695,E2 -7088.695} C_VEL
LIN {X 0,Y 473.755,Z 374.901,A -85,B 0,C 180,E1 -7090.049,E2 -7090.049} C_VEL
LIN {X 0,Y 473.677,Z 377.404,A -85,B 0,C 180,E1 -7091.844,E2 -7091.844} C_VEL
LIN {X 0,Y 473.593,Z 378.436,A -85,B 0,C 180,E1 -7093.622,E2 -7093.622} C_VEL
LIN {X 0,Y 473.642,Z 378.044,A -85,B 0,C 180,E1 -7095.388,E2 -7095.388} C_VEL
LIN {X 0,Y 473.685,Z 376.255,A -85,B 0,C 180,E1 -7097.14,E2 -7097.14} C_VEL
LIN {X 0,Y 473.81,Z 373.053,A -85,B 0,C 180,E1 -7098.881,E2 -7098.881} C_VEL
LIN {X 0,Y 473.909,Z 369.637,A -85,B 0,C 180,E1 -7100.179,E2 -7100.179} C_VEL
LIN {X 0,Y 474.14,Z 363.739,A -85,B 0,C 180,E1 -7101.904,E2 -7101.904} C_VEL
LIN {X 0,Y 474.467,Z 357.107,A -85,B 0,C 180,E1 -7103.407,E2 -7103.407} C_VEL
LIN {X 0,Y 474.838,Z 348.891,A -85,B 0,C 180,E1 -7104.904,E2 -7104.904} C_VEL
LIN {X 0,Y 475.306,Z 340.336,A -85,B 0,C 180,E1 -7106.184,E2 -7106.184} C_VEL
LIN {X 0,Y 475.853,Z 330.012,A -85,B 0,C 180,E1 -7107.459,E2 -7107.459} C_VEL
LIN {X 0,Y 476.402,Z 319.66,A -85,B 0,C 180,E1 -7108.519,E2 -7108.519} C_VEL
LIN {X 0,Y 476.976,Z 308.421,A -85,B 0,C 180,E1 -7109.471,E2 -7109.471} C_VEL
LIN {X 0,Y 477.65,Z 296.096,A -85,B 0,C 180,E1 -7110.315,E2 -7110.315} C_VEL
LIN {X 0,Y 478.155,Z 283.22,A -85,B 0,C 180,E1 -7111.015,E2 -7111.015} C_VEL
LIN {X 0,Y 478.558,Z 268.985,A -85,B 0,C 180,E1 -7111.597,E2 -7111.597} C_VEL
LIN {X 0,Y 478.86,Z 254.686,A -85,B 0,C 180,E1 -7111.996,E2 -7111.996} C_VEL
LIN {X 0,Y 479.538,Z 190.386,A -85,B 0,C 180,E1 -7112.997,E2 -7112.997} C_VEL
LIN {X 0,Y 480.027,Z 133.812,A -85,B 0,C 180,E1 -7113.859,E2 -7113.859} C_VEL
LIN {X 0,Y 476.556,Z 117.137,A -85,B 0,C 180,E1 -7114.28,E2 -7114.28} C_VEL
LIN {X 0,Y 476.883,Z 108.188,A -85,B 0,C 180,E1 -7115.92,E2 -7115.92} C_VEL
LIN {X 0,Y 474.748,Z 96.976,A -85,B 0,C 180,E1 -7118.158,E2 -7118.158} C_VEL
LIN {X 0,Y 474.702,Z 96.984,A -85,B 0,C 180,E1 -7121.961,E2 -7121.961} C_VEL
LIN {X 0,Y 474.686,Z 96.982,A -85,B 0,C 180,E1 -7125.455,E2 -7125.455} C_VEL
LIN {X 0,Y 474.634,Z 96.983,A -85,B 0,C 180,E1 -7128.634,E2 -7128.634} C_VEL
LIN {X 0,Y 474.61,Z 96.991,A -85,B 0,C 180,E1 -7131.726,E2 -7131.726} C_VEL
LIN {X 0,Y 474.641,Z 96.982,A -85,B 0,C 180,E1 -7134.492,E2 -7134.492} C_VEL
LIN {X 0,Y 474.661,Z 96.987,A -85,B 0,C 180,E1 -7137.34,E2 -7137.34} C_VEL
LIN {X 0,Y 474.587,Z 96.992,A -85,B 0,C 180,E1 -7140.815,E2 -7140.815} C_VEL
LIN {X 0,Y 474.605,Z 96.987,A -85,B 0,C 180,E1 -7143.986,E2 -7143.986} C_VEL
LIN {X 0,Y 474.557,Z 96.999,A -85,B 0,C 180,E1 -7146.904,E2 -7146.904} C_VEL
LIN {X 0,Y 474.638,Z 96.983,A -85,B 0,C 180,E1 -7149.656,E2 -7149.656} C_VEL
LIN {X 0,Y 474.629,Z 96.99,A -85,B 0,C 180,E1 -7152.931,E2 -7152.931} C_VEL
LIN {X 0,Y 474.644,Z 96.982,A -85,B 0,C 180,E1 -7155.905,E2 -7155.905} C_VEL
LIN {X 0,Y 474.618,Z 96.988,A -85,B 0,C 180,E1 -7159.04,E2 -7159.04} C_VEL
LIN {X 0,Y 474.593,Z 96.988,A -85,B 0,C 180,E1 -7161.704,E2 -7161.704} C_VEL
LIN {X 0,Y 474.605,Z 96.991,A -85,B 0,C 180,E1 -7164.729,E2 -7164.729} C_VEL
LIN {X 0,Y 474.613,Z 96.987,A -85,B 0,C 180,E1 -7167.791,E2 -7167.791} C_VEL
LIN {X 0,Y 474.607,Z 96.987,A -85,B 0,C 180,E1 -7170.885,E2 -7170.885} C_VEL
LIN {X 0,Y 474.644,Z 96.983,A -85,B 0,C 180,E1 -7173.632,E2 -7173.632} C_VEL
LIN {X 0,Y 474.632,Z 96.985,A -85,B 0,C 180,E1 -7176.639,E2 -7176.639} C_VEL
LIN {X 0,Y 474.656,Z 96.981,A -85,B 0,C 180,E1 -7179.188,E2 -7179.188} C_VEL
LIN {X 0,Y 474.638,Z 96.991,A -85,B 0,C 180,E1 -7181.887,E2 -7181.887} C_VEL
LIN {X 0,Y 474.682,Z 96.978,A -85,B 0,C 180,E1 -7184.547,E2 -7184.547} C_VEL
LIN {X 0,Y 474.723,Z 96.976,A -85,B 0,C 180,E1 -7188.041,E2 -7188.041} C_VEL
LIN {X 0,Y 474.715,Z 96.979,A -85,B 0,C 180,E1 -7191.489,E2 -7191.489} C_VEL
LIN {X 0,Y 474.772,Z 96.968,A -85,B 0,C 180,E1 -7194.055,E2 -7194.055} C_VEL
LIN {X 0,Y 474.884,Z 96.96,A -85,B 0,C 180,E1 -7197.458,E2 -7197.458} C_VEL
LIN {X 0,Y 474.868,Z 96.956,A -85,B 0,C 180,E1 -7200.851,E2 -7200.851} C_VEL
LIN {X 0,Y 474.885,Z 96.952,A -85,B 0,C 180,E1 -7202.547,E2 -7202.547} C_VEL
LIN {X 0,Y 474.771,Z 96.966,A -85,B 0,C 180,E1 -7205.95,E2 -7205.95} C_VEL
LIN {X 0,Y 474.72,Z 96.974,A -85,B 0,C 180,E1 -7208.516,E2 -7208.516} C_VEL
LIN {X 0,Y 474.697,Z 96.975,A -85,B 0,C 180,E1 -7211.965,E2 -7211.965} C_VEL
LIN {X 0,Y 474.694,Z 96.977,A -85,B 0,C 180,E1 -7215.458,E2 -7215.458} C_VEL
LIN {X 0,Y 474.659,Z 96.985,A -85,B 0,C 180,E1 -7219.013,E2 -7219.013} C_VEL
LIN {X 0,Y 474.585,Z 96.989,A -85,B 0,C 180,E1 -7221.731,E2 -7221.731} C_VEL
LIN {X 0,Y 474.655,Z 96.987,A -85,B 0,C 180,E1 -7224.495,E2 -7224.495} C_VEL
LIN {X 0,Y 474.696,Z 96.976,A -85,B 0,C 180,E1 -7227.341,E2 -7227.341} C_VEL
LIN {X 0,Y 474.601,Z 96.99,A -85,B 0,C 180,E1 -7230.812,E2 -7230.812} C_VEL
LIN {X 0,Y 474.636,Z 96.987,A -85,B 0,C 180,E1 -7233.986,E2 -7233.986} C_VEL
LIN {X 0,Y 474.572,Z 96.992,A -85,B 0,C 180,E1 -7236.902,E2 -7236.902} C_VEL
LIN {X 0,Y 474.625,Z 96.986,A -85,B 0,C 180,E1 -7239.65,E2 -7239.65} C_VEL
LIN {X 0,Y 474.614,Z 96.986,A -85,B 0,C 180,E1 -7242.936,E2 -7242.936} C_VEL
LIN {X 0,Y 474.607,Z 96.994,A -85,B 0,C 180,E1 -7245.897,E2 -7245.897} C_VEL
LIN {X 0,Y 474.627,Z 96.984,A -85,B 0,C 180,E1 -7249.043,E2 -7249.043} C_VEL
LIN {X 0,Y 474.61,Z 96.994,A -85,B 0,C 180,E1 -7251.706,E2 -7251.706} C_VEL
LIN {X 0,Y 474.624,Z 96.984,A -85,B 0,C 180,E1 -7254.727,E2 -7254.727} C_VEL
LIN {X 0,Y 474.636,Z 96.99,A -85,B 0,C 180,E1 -7257.789,E2 -7257.789} C_VEL
LIN {X 0,Y 474.624,Z 96.991,A -85,B 0,C 180,E1 -7260.887,E2 -7260.887} C_VEL
LIN {X 0,Y 474.689,Z 96.993,A -85,B 0,C 180,E1 -7262.547,E2 -7262.547} C_VEL
LIN {X 0,Y 477.56,Z 110.895,A -85,B 0,C 180,E1 -7264.971,E2 -7264.971} C_VEL
LIN {X 0,Y 477.146,Z 122.346,A -85,B 0,C 180,E1 -7266.797,E2 -7266.797} C_VEL
LIN {X 0,Y 476.344,Z 141.133,A -85,B 0,C 180,E1 -7269.754,E2 -7269.754} C_VEL
LIN {X 0,Y 479.909,Z 162.112,A -85,B 0,C 180,E1 -7270.226,E2 -7270.226} C_VEL
LIN {X 0,Y 478.781,Z 279.112,A -85,B 0,C 180,E1 -7272.019,E2 -7272.019} C_VEL
LIN {X 0,Y 478.371,Z 294.024,A -85,B 0,C 180,E1 -7272.426,E2 -7272.426} C_VEL
LIN {X 0,Y 477.932,Z 307.558,A -85,B 0,C 180,E1 -7272.968,E2 -7272.968} C_VEL
LIN {X 0,Y 477.348,Z 320.678,A -85,B 0,C 180,E1 -7273.664,E2 -7273.664} C_VEL
LIN {X 0,Y 476.74,Z 333.108,A -85,B 0,C 180,E1 -7274.504,E2 -7274.504} C_VEL
LIN {X 0,Y 476.072,Z 344.688,A -85,B 0,C 180,E1 -7275.467,E2 -7275.467} C_VEL
LIN {X 0,Y 475.53,Z 355.314,A -85,B 0,C 180,E1 -7276.541,E2 -7276.541} C_VEL
LIN {X 0,Y 475.042,Z 366.005,A -85,B 0,C 180,E1 -7277.849,E2 -7277.849} C_VEL
LIN {X 0,Y 474.578,Z 374.565,A -85,B 0,C 180,E1 -7279.118,E2 -7279.118} C_VEL
LIN {X 0,Y 474.23,Z 382.903,A -85,B 0,C 180,E1 -7280.619,E2 -7280.619} C_VEL
LIN {X 0,Y 473.991,Z 388.716,A -85,B 0,C 180,E1 -7281.904,E2 -7281.904} C_VEL
LIN {X 0,Y 473.894,Z 393.493,A -85,B 0,C 180,E1 -7283.187,E2 -7283.187} C_VEL
LIN {X 0,Y 473.815,Z 398.433,A -85,B 0,C 180,E1 -7284.895,E2 -7284.895} C_VEL
LIN {X 0,Y 473.756,Z 401.867,A -85,B 0,C 180,E1 -7286.599,E2 -7286.599} C_VEL
LIN {X 0,Y 473.697,Z 403.899,A -85,B 0,C 180,E1 -7288.301,E2 -7288.301} C_VEL
LIN {X 0,Y 473.672,Z 404.578,A -85,B 0,C 180,E1 -7290.001,E2 -7290.001} C_VEL
LIN {X 0,Y 473.697,Z 403.915,A -85,B 0,C 180,E1 -7291.702,E2 -7291.702} C_VEL
LIN {X 0,Y 473.757,Z 401.901,A -85,B 0,C 180,E1 -7293.403,E2 -7293.403} C_VEL
LIN {X 0,Y 473.816,Z 398.487,A -85,B 0,C 180,E1 -7295.107,E2 -7295.107} C_VEL
LIN {X 0,Y 473.895,Z 393.576,A -85,B 0,C 180,E1 -7296.815,E2 -7296.815} C_VEL
LIN {X 0,Y 474.071,Z 387.025,A -85,B 0,C 180,E1 -7298.527,E2 -7298.527} C_VEL
LIN {X 0,Y 474.342,Z 379.743,A -85,B 0,C 180,E1 -7300.027,E2 -7300.027} C_VEL
LIN {X 0,Y 474.842,Z 370.744,A -85,B 0,C 180,E1 -7301.527,E2 -7301.527} C_VEL
LIN {X 0,Y 475.291,Z 361.305,A -85,B 0,C 180,E1 -7302.816,E2 -7302.816} C_VEL
LIN {X 0,Y 475.895,Z 349.805,A -85,B 0,C 180,E1 -7304.104,E2 -7304.104} C_VEL
LIN {X 0,Y 476.536,Z 338.112,A -85,B 0,C 180,E1 -7305.177,E2 -7305.177} C_VEL
LIN {X 0,Y 477.279,Z 325.126,A -85,B 0,C 180,E1 -7306.138,E2 -7306.138} C_VEL
LIN {X 0,Y 477.945,Z 311.387,A -85,B 0,C 180,E1 -7306.939,E2 -7306.939} C_VEL
LIN {X 0,Y 478.491,Z 297.619,A -85,B 0,C 180,E1 -7307.541,E2 -7307.541} C_VEL
LIN {X 0,Y 478.913,Z 283.496,A -85,B 0,C 180,E1 -7307.978,E2 -7307.978} C_VEL
LIN {X 0,Y 479.279,Z 266.243,A -85,B 0,C 180,E1 -7308.295,E2 -7308.295} C_VEL
LIN {X 0,Y 480.149,Z 161.058,A -85,B 0,C 180,E1 -7309.914,E2 -7309.914} C_VEL
LIN {X 0,Y 476.465,Z 140.882,A -85,B 0,C 180,E1 -7310.414,E2 -7310.414} C_VEL
LIN {X 0,Y 477.466,Z 120.954,A -85,B 0,C 180,E1 -7313.608,E2 -7313.608} C_VEL
LIN {X 0,Y 477.934,Z 112.34,A -85,B 0,C 180,E1 -7315.011,E2 -7315.011} C_VEL
LIN {X 0,Y 475.13,Z 99.024,A -85,B 0,C 180,E1 -7317.437,E2 -7317.437} C_VEL
LIN {X 0,Y 474.672,Z 96.983,A -85,B 0,C 180,E1 -7317.861,E2 -7317.861} C_VEL
LIN {X 0,Y 474.609,Z 96.994,A -85,B 0,C 180,E1 -7321.218,E2 -7321.218} C_VEL
LIN {X 0,Y 474.631,Z 96.99,A -85,B 0,C 180,E1 -7324.242,E2 -7324.242} C_VEL
LIN {X 0,Y 474.596,Z 96.989,A -85,B 0,C 180,E1 -7327.384,E2 -7327.384} C_VEL
LIN {X 0,Y 474.627,Z 96.984,A -85,B 0,C 180,E1 -7330.658,E2 -7330.658} C_VEL
LIN {X 0,Y 474.603,Z 96.99,A -85,B 0,C 180,E1 -7333.479,E2 -7333.479} C_VEL
LIN {X 0,Y 474.608,Z 96.989,A -85,B 0,C 180,E1 -7336.519,E2 -7336.519} C_VEL
LIN {X 0,Y 474.628,Z 96.978,A -85,B 0,C 180,E1 -7339.341,E2 -7339.341} C_VEL
LIN {X 0,Y 474.597,Z 96.987,A -85,B 0,C 180,E1 -7342.615,E2 -7342.615} C_VEL
LIN {X 0,Y 474.633,Z 96.987,A -85,B 0,C 180,E1 -7345.757,E2 -7345.757} C_VEL
LIN {X 0,Y 474.611,Z 96.987,A -85,B 0,C 180,E1 -7348.781,E2 -7348.781} C_VEL
LIN {X 0,Y 474.632,Z 96.983,A -85,B 0,C 180,E1 -7351.715,E2 -7351.715} C_VEL
LIN {X 0,Y 474.664,Z 96.982,A -85,B 0,C 180,E1 -7354.581,E2 -7354.581} C_VEL
LIN {X 0,Y 474.613,Z 96.991,A -85,B 0,C 180,E1 -7357.354,E2 -7357.354} C_VEL
LIN {X 0,Y 474.665,Z 96.976,A -85,B 0,C 180,E1 -7360.088,E2 -7360.088} C_VEL
LIN {X 0,Y 474.647,Z 96.987,A -85,B 0,C 180,E1 -7362.772,E2 -7362.772} C_VEL
LIN {X 0,Y 474.653,Z 96.982,A -85,B 0,C 180,E1 -7365.419,E2 -7365.419} C_VEL
LIN {X 0,Y 474.716,Z 96.973,A -85,B 0,C 180,E1 -7368.035,E2 -7368.035} C_VEL
LIN {X 0,Y 474.718,Z 96.972,A -85,B 0,C 180,E1 -7371.484,E2 -7371.484} C_VEL
LIN {X 0,Y 474.75,Z 96.971,A -85,B 0,C 180,E1 -7374.902,E2 -7374.902} C_VEL
LIN {X 0,Y 474.893,Z 96.948,A -85,B 0,C 180,E1 -7377.453,E2 -7377.453} C_VEL
LIN {X 0,Y 474.917,Z 96.955,A -85,B 0,C 180,E1 -7379.997,E2 -7379.997} C_VEL
LIN {X 0,Y 474.891,Z 96.954,A -85,B 0,C 180,E1 -7382.542,E2 -7382.542} C_VEL
LIN {X 0,Y 474.762,Z 96.971,A -85,B 0,C 180,E1 -7385.945,E2 -7385.945} C_VEL
LIN {X 0,Y 474.715,Z 96.973,A -85,B 0,C 180,E1 -7388.511,E2 -7388.511} C_VEL
LIN {X 0,Y 474.706,Z 96.978,A -85,B 0,C 180,E1 -7391.959,E2 -7391.959} C_VEL
LIN {X 0,Y 474.699,Z 96.983,A -85,B 0,C 180,E1 -7395.452,E2 -7395.452} C_VEL
LIN {X 0,Y 474.659,Z 96.984,A -85,B 0,C 180,E1 -7399.007,E2 -7399.007} C_VEL
LIN {X 0,Y 474.584,Z 96.993,A -85,B 0,C 180,E1 -7401.725,E2 -7401.725} C_VEL
LIN {X 0,Y 474.623,Z 96.986,A -85,B 0,C 180,E1 -7404.491,E2 -7404.491} C_VEL
LIN {X 0,Y 474.666,Z 96.985,A -85,B 0,C 180,E1 -7407.329,E2 -7407.329} C_VEL
LIN {X 0,Y 474.594,Z 96.981,A -85,B 0,C 180,E1 -7410.227,E2 -7410.227} C_VEL
LIN {X 0,Y 474.613,Z 96.986,A -85,B 0,C 180,E1 -7413.218,E2 -7413.218} C_VEL
LIN {X 0,Y 474.575,Z 96.996,A -85,B 0,C 180,E1 -7416.32,E2 -7416.32} C_VEL
LIN {X 0,Y 474.599,Z 96.991,A -85,B 0,C 180,E1 -7419.642,E2 -7419.642} C_VEL
LIN {X 0,Y 474.607,Z 96.992,A -85,B 0,C 180,E1 -7422.233,E2 -7422.233} C_VEL
LIN {X 0,Y 474.596,Z 96.989,A -85,B 0,C 180,E1 -7425.294,E2 -7425.294} C_VEL
LIN {X 0,Y 474.592,Z 97.002,A -85,B 0,C 180,E1 -7428.21,E2 -7428.21} C_VEL
LIN {X 0,Y 474.641,Z 97.163,A -85,B 0,C 180,E1 -7429.632,E2 -7429.632} C_VEL
LIN {X 0,Y 477.015,Z 108.836,A -85,B 0,C 180,E1 -7432.031,E2 -7432.031} C_VEL
LIN {X 0,Y 476.759,Z 117.503,A -85,B 0,C 180,E1 -7433.658,E2 -7433.658} C_VEL
LIN {X 0,Y 480.434,Z 134.095,A -85,B 0,C 180,E1 -7434.102,E2 -7434.102} C_VEL
LIN {X 0,Y 479.253,Z 253.554,A -85,B 0,C 180,E1 -7435.954,E2 -7435.954} C_VEL
LIN {X 0,Y 478.512,Z 257.458,A -85,B 0,C 180,E1 -7436.01,E2 -7436.01} C_VEL
LIN {X 0,Y 472.769,Z 269.64,A -85,B 0,C 180,E1 -7436.141,E2 -7436.141} C_VEL
LIN {X 0,Y 472.044,Z 273.44,A -85,B 0,C 180,E1 -7436.253,E2 -7436.253} C_VEL
LIN {X 0,Y 471.556,Z 286.707,A -85,B 0,C 180,E1 -7436.852,E2 -7436.852} C_VEL
LIN {X 0,Y 470.909,Z 299.807,A -85,B 0,C 180,E1 -7437.627,E2 -7437.627} C_VEL
LIN {X 0,Y 470.174,Z 312.508,A -85,B 0,C 180,E1 -7438.579,E2 -7438.579} C_VEL
LIN {X 0,Y 469.506,Z 324.092,A -85,B 0,C 180,E1 -7439.654,E2 -7439.654} C_VEL
LIN {X 0,Y 468.853,Z 334.642,A -85,B 0,C 180,E1 -7440.844,E2 -7440.844} C_VEL
LIN {X 0,Y 468.182,Z 345.004,A -85,B 0,C 180,E1 -7442.266,E2 -7442.266} C_VEL
LIN {X 0,Y 467.678,Z 353.432,A -85,B 0,C 180,E1 -7443.684,E2 -7443.684} C_VEL
LIN {X 0,Y 467.31,Z 360.298,A -85,B 0,C 180,E1 -7445.095,E2 -7445.095} C_VEL
LIN {X 0,Y 467.03,Z 366.287,A -85,B 0,C 180,E1 -7446.616,E2 -7446.616} C_VEL
LIN {X 0,Y 466.863,Z 371.553,A -85,B 0,C 180,E1 -7448.356,E2 -7448.356} C_VEL
LIN {X 0,Y 466.7,Z 374.647,A -85,B 0,C 180,E1 -7449.734,E2 -7449.734} C_VEL
LIN {X 0,Y 466.594,Z 377.382,A -85,B 0,C 180,E1 -7451.559,E2 -7451.559} C_VEL
LIN {X 0,Y 466.502,Z 378.589,A -85,B 0,C 180,E1 -7453.366,E2 -7453.366} C_VEL
LIN {X 0,Y 466.547,Z 378.37,A -85,B 0,C 180,E1 -7455.161,E2 -7455.161} C_VEL
LIN {X 0,Y 466.577,Z 376.753,A -85,B 0,C 180,E1 -7456.94,E2 -7456.94} C_VEL
LIN {X 0,Y 466.724,Z 373.724,A -85,B 0,C 180,E1 -7458.71,E2 -7458.71} C_VEL
LIN {X 0,Y 466.852,Z 369.238,A -85,B 0,C 180,E1 -7460.467,E2 -7460.467} C_VEL
LIN {X 0,Y 467.036,Z 364.784,A -85,B 0,C 180,E1 -7461.78,E2 -7461.78} C_VEL
LIN {X 0,Y 467.333,Z 358.728,A -85,B 0,C 180,E1 -7463.227,E2 -7463.227} C_VEL
LIN {X 0,Y 467.658,Z 351.64,A -85,B 0,C 180,E1 -7464.609,E2 -7464.609} C_VEL
LIN {X 0,Y 468.128,Z 343.584,A -85,B 0,C 180,E1 -7465.909,E2 -7465.909} C_VEL
LIN {X 0,Y 468.678,Z 333.907,A -85,B 0,C 180,E1 -7467.205,E2 -7467.205} C_VEL
LIN {X 0,Y 469.298,Z 323.195,A -85,B 0,C 180,E1 -7468.39,E2 -7468.39} C_VEL
LIN {X 0,Y 469.971,Z 311.346,A -85,B 0,C 180,E1 -7469.463,E2 -7469.463} C_VEL
LIN {X 0,Y 470.617,Z 299.692,A -85,B 0,C 180,E1 -7470.32,E2 -7470.32} C_VEL
LIN {X 0,Y 471.158,Z 286.906,A -85,B 0,C 180,E1 -7471.075,E2 -7471.075} C_VEL
LIN {X 0,Y 471.683,Z 272.779,A -85,B 0,C 180,E1 -7471.706,E2 -7471.706} C_VEL
LIN {X 0,Y 472.021,Z 258.302,A -85,B 0,C 180,E1 -7472.159,E2 -7472.159} C_VEL
LIN {X 0,Y 472.272,Z 241.206,A -85,B 0,C 180,E1 -7472.478,E2 -7472.478} C_VEL
LIN {X 0,Y 473.235,Z 134.613,A -85,B 0,C 180,E1 -7474.122,E2 -7474.122} C_VEL
LIN {X 0,Y 469.66,Z 117.357,A -85,B 0,C 180,E1 -7474.558,E2 -7474.558} C_VEL
LIN {X 0,Y 469.937,Z 109.561,A -85,B 0,C 180,E1 -7476.008,E2 -7476.008} C_VEL
LIN {X 0,Y 467.697,Z 97.854,A -85,B 0,C 180,E1 -7478.372,E2 -7478.372} C_VEL
LIN {X 0,Y 467.66,Z 97.862,A -85,B 0,C 180,E1 -7482.144,E2 -7482.144} C_VEL
LIN {X 0,Y 467.606,Z 97.859,A -85,B 0,C 180,E1 -7484.802,E2 -7484.802} C_VEL
LIN {X 0,Y 467.588,Z 97.867,A -85,B 0,C 180,E1 -7487.493,E2 -7487.493} C_VEL
LIN {X 0,Y 467.589,Z 97.861,A -85,B 0,C 180,E1 -7490.223,E2 -7490.223} C_VEL
LIN {X 0,Y 467.571,Z 97.869,A -85,B 0,C 180,E1 -7493.537,E2 -7493.537} C_VEL
LIN {X 0,Y 467.582,Z 97.864,A -85,B 0,C 180,E1 -7495.84,E2 -7495.84} C_VEL
LIN {X 0,Y 467.548,Z 97.868,A -85,B 0,C 180,E1 -7498.75,E2 -7498.75} C_VEL
LIN {X 0,Y 467.558,Z 97.866,A -85,B 0,C 180,E1 -7501.74,E2 -7501.74} C_VEL
LIN {X 0,Y 467.544,Z 97.871,A -85,B 0,C 180,E1 -7504.833,E2 -7504.833} C_VEL
LIN {X 0,Y 467.566,Z 97.864,A -85,B 0,C 180,E1 -7508.043,E2 -7508.043} C_VEL
LIN {X 0,Y 467.57,Z 97.864,A -85,B 0,C 180,E1 -7510.263,E2 -7510.263} C_VEL
LIN {X 0,Y 467.586,Z 97.866,A -85,B 0,C 180,E1 -7512.573,E2 -7512.573} C_VEL
LIN {X 0,Y 467.606,Z 97.861,A -85,B 0,C 180,E1 -7516.267,E2 -7516.267} C_VEL
LIN {X 0,Y 467.572,Z 97.863,A -85,B 0,C 180,E1 -7519.74,E2 -7519.74} C_VEL
LIN {X 0,Y 467.527,Z 97.872,A -85,B 0,C 180,E1 -7522.815,E2 -7522.815} C_VEL
LIN {X 0,Y 467.56,Z 97.87,A -85,B 0,C 180,E1 -7526.214,E2 -7526.214} C_VEL
LIN {X 0,Y 467.55,Z 97.865,A -85,B 0,C 180,E1 -7529.269,E2 -7529.269} C_VEL
LIN {X 0,Y 467.621,Z 97.861,A -85,B 0,C 180,E1 -7532.461,E2 -7532.461} C_VEL
LIN {X 0,Y 467.595,Z 97.86,A -85,B 0,C 180,E1 -7535.116,E2 -7535.116} C_VEL
LIN {X 0,Y 467.558,Z 97.871,A -85,B 0,C 180,E1 -7537.931,E2 -7537.931} C_VEL
LIN {X 0,Y 467.604,Z 97.859,A -85,B 0,C 180,E1 -7540.695,E2 -7540.695} C_VEL
LIN {X 0,Y 467.648,Z 97.858,A -85,B 0,C 180,E1 -7544.11,E2 -7544.11} C_VEL
LIN {X 0,Y 467.667,Z 97.857,A -85,B 0,C 180,E1 -7547.858,E2 -7547.858} C_VEL
LIN {X 0,Y 467.669,Z 97.855,A -85,B 0,C 180,E1 -7551.36,E2 -7551.36} C_VEL
LIN {X 0,Y 467.735,Z 97.845,A -85,B 0,C 180,E1 -7553.966,E2 -7553.966} C_VEL
LIN {X 0,Y 467.85,Z 97.836,A -85,B 0,C 180,E1 -7557.42,E2 -7557.42} C_VEL
LIN {X 0,Y 467.871,Z 97.826,A -85,B 0,C 180,E1 -7560.003,E2 -7560.003} C_VEL
LIN {X 0,Y 467.851,Z 97.829,A -85,B 0,C 180,E1 -7562.586,E2 -7562.586} C_VEL
LIN {X 0,Y 467.735,Z 97.843,A -85,B 0,C 180,E1 -7566.04,E2 -7566.04} C_VEL
LIN {X 0,Y 467.674,Z 97.853,A -85,B 0,C 180,E1 -7568.645,E2 -7568.645} C_VEL
LIN {X 0,Y 467.649,Z 97.853,A -85,B 0,C 180,E1 -7572.148,E2 -7572.148} C_VEL
LIN {X 0,Y 467.633,Z 97.855,A -85,B 0,C 180,E1 -7575.698,E2 -7575.698} C_VEL
LIN {X 0,Y 467.612,Z 97.866,A -85,B 0,C 180,E1 -7578.767,E2 -7578.767} C_VEL
LIN {X 0,Y 467.576,Z 97.864,A -85,B 0,C 180,E1 -7581.271,E2 -7581.271} C_VEL
LIN {X 0,Y 467.569,Z 97.864,A -85,B 0,C 180,E1 -7583.946,E2 -7583.946} C_VEL
LIN {X 0,Y 467.625,Z 97.86,A -85,B 0,C 180,E1 -7586.802,E2 -7586.802} C_VEL
LIN {X 0,Y 467.551,Z 97.866,A -85,B 0,C 180,E1 -7589.74,E2 -7589.74} C_VEL
LIN {X 0,Y 467.581,Z 97.864,A -85,B 0,C 180,E1 -7592.761,E2 -7592.761} C_VEL
LIN {X 0,Y 467.554,Z 97.869,A -85,B 0,C 180,E1 -7595.892,E2 -7595.892} C_VEL
LIN {X 0,Y 467.58,Z 97.862,A -85,B 0,C 180,E1 -7599.147,E2 -7599.147} C_VEL
